FUNCTION "AHUTemperatureDemand" : Void   // FC60007, LAD
{ S7_Optimized_Access := 'TRUE' }
VERSION : 0.1
// stored: AutoNumber false, IsIECCheckEnabled false, SetENOAutomatically false, UDAEnableTagReadback false
   VAR_INPUT
      iUnitID : Int;
      cCoolingRegulatorState : Byte;
      cHeatingRegulatorState : Byte;
      rSATActual : Real;
      rSATSP : Real;
      rRATActual : Real;
      rRATSPHeating : Real;
      rRATSPCooling : Real;
   END_VAR
   VAR_OUTPUT
      rHeatingDemand : Real;
      rCoolingDemand : Real;
      rFreshAirTempDemand : Real;
   END_VAR
   VAR_TEMP
      iActualUnitMode_old : Int;
      xResetActualSetpoints : Bool;
   END_VAR
   VAR CONSTANT
      cZero : Byte;
   END_VAR
   VAR_TEMP   // added for the SCL form of the ladder/FBD networks
      _w1 : Bool;
   END_VAR
BEGIN

REGION Network 1: Cooling
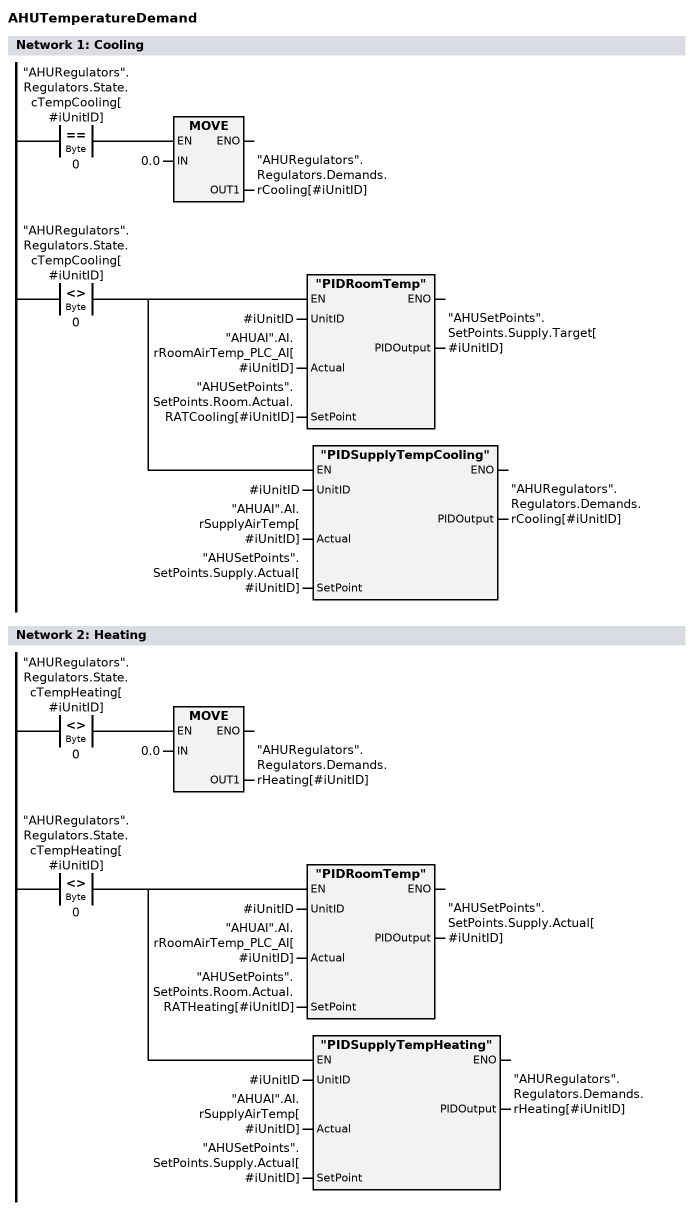
   RUNG wire#powerrail
      { S7_Templates := "SrcType := Byte" } EQ_Contact(in1 := "AHURegulators".Regulators.State.cTempCooling[#iUnitID], in2 := 0)
      Move(in := 0.0, out1 => "AHURegulators".Regulators.Demands.rCooling[#iUnitID])
   END_RUNG
   RUNG wire#powerrail
      { S7_Templates := "SrcType := Byte" } NE_Contact(in1 := "AHURegulators".Regulators.State.cTempCooling[#iUnitID], in2 := 0)
      wire#w1
      "PIDRoomTemp"(UnitID := #iUnitID, Actual := "AHUAI".AI.rRoomAirTemp_PLC_AI[#iUnitID], SetPoint := "AHUSetPoints".SetPoints.Room.Actual.RATCooling[#iUnitID], PIDOutput => "AHUSetPoints".SetPoints.Supply.Target[#iUnitID])
   END_RUNG
   RUNG wire#w1
      "PIDSupplyTempCooling"(UnitID := #iUnitID, Actual := "AHUAI".AI.rSupplyAirTemp[#iUnitID], SetPoint := "AHUSetPoints".SetPoints.Supply.Actual[#iUnitID], PIDOutput => "AHURegulators".Regulators.Demands.rCooling[#iUnitID])
   END_RUNG
   // the same network as SCL:
   IF "AHURegulators".Regulators.State.cTempCooling[#iUnitID] = 0 THEN
       "AHURegulators".Regulators.Demands.rCooling[#iUnitID] := 0.0;
   END_IF;
   #_w1 := "AHURegulators".Regulators.State.cTempCooling[#iUnitID] <> 0;
   IF #_w1 THEN
       "PIDRoomTemp"(UnitID := #iUnitID,
                     Actual := "AHUAI".AI.rRoomAirTemp_PLC_AI[#iUnitID],
                     SetPoint := "AHUSetPoints".SetPoints.Room.Actual.RATCooling[#iUnitID],
                     PIDOutput => "AHUSetPoints".SetPoints.Supply.Target[#iUnitID]);
       "PIDSupplyTempCooling"(UnitID := #iUnitID,
                              Actual := "AHUAI".AI.rSupplyAirTemp[#iUnitID],
                              SetPoint := "AHUSetPoints".SetPoints.Supply.Actual[#iUnitID],
                              PIDOutput => "AHURegulators".Regulators.Demands.rCooling[#iUnitID]);
   END_IF;
END_REGION

REGION Network 2: Heating
   RUNG wire#powerrail
      { S7_Templates := "SrcType := Byte" } NE_Contact(in1 := "AHURegulators".Regulators.State.cTempHeating[#iUnitID], in2 := 0)
      Move(in := 0.0, out1 => "AHURegulators".Regulators.Demands.rHeating[#iUnitID])
   END_RUNG
   RUNG wire#powerrail
      { S7_Templates := "SrcType := Byte" } NE_Contact(in1 := "AHURegulators".Regulators.State.cTempHeating[#iUnitID], in2 := 0)
      wire#w1
      "PIDRoomTemp"(UnitID := #iUnitID, Actual := "AHUAI".AI.rRoomAirTemp_PLC_AI[#iUnitID], SetPoint := "AHUSetPoints".SetPoints.Room.Actual.RATHeating[#iUnitID], PIDOutput => "AHUSetPoints".SetPoints.Supply.Actual[#iUnitID])
   END_RUNG
   RUNG wire#w1
      "PIDSupplyTempHeating"(UnitID := #iUnitID, Actual := "AHUAI".AI.rSupplyAirTemp[#iUnitID], SetPoint := "AHUSetPoints".SetPoints.Supply.Actual[#iUnitID], PIDOutput => "AHURegulators".Regulators.Demands.rHeating[#iUnitID])
   END_RUNG
   // the same network as SCL:
   IF "AHURegulators".Regulators.State.cTempHeating[#iUnitID] <> 0 THEN
       "AHURegulators".Regulators.Demands.rHeating[#iUnitID] := 0.0;
   END_IF;
   #_w1 := "AHURegulators".Regulators.State.cTempHeating[#iUnitID] <> 0;
   IF #_w1 THEN
       "PIDRoomTemp"(UnitID := #iUnitID,
                     Actual := "AHUAI".AI.rRoomAirTemp_PLC_AI[#iUnitID],
                     SetPoint := "AHUSetPoints".SetPoints.Room.Actual.RATHeating[#iUnitID],
                     PIDOutput => "AHUSetPoints".SetPoints.Supply.Actual[#iUnitID]);
       "PIDSupplyTempHeating"(UnitID := #iUnitID,
                              Actual := "AHUAI".AI.rSupplyAirTemp[#iUnitID],
                              SetPoint := "AHUSetPoints".SetPoints.Supply.Actual[#iUnitID],
                              PIDOutput => "AHURegulators".Regulators.Demands.rHeating[#iUnitID]);
   END_IF;
END_REGION
END_FUNCTION

FUNCTION "PIDRoomTemp" : Void   // FC8, FBD
{ S7_Optimized_Access := 'TRUE' }
VERSION : 0.1
// stored: AutoNumber false, IsIECCheckEnabled false, SetENOAutomatically false, UDAEnableTagReadback false
   VAR_INPUT
      UnitID : Int;
      Actual : Real;
      SetPoint : Real;
   END_VAR
   VAR_OUTPUT
      PIDOutput : Real;
   END_VAR
BEGIN
END_FUNCTION

FUNCTION "PIDSupplyTempCooling" : Void   // FC12, FBD
{ S7_Optimized_Access := 'TRUE' }
VERSION : 0.1
// stored: AutoNumber false, IsIECCheckEnabled false, SetENOAutomatically false, UDAEnableTagReadback false
   VAR_INPUT
      UnitID : Int;
      Actual : Real;
      SetPoint : Real;
   END_VAR
   VAR_OUTPUT
      PIDOutput : Real;
   END_VAR
BEGIN
END_FUNCTION

FUNCTION "PIDSupplyTempHeating" : Void   // FC10, FBD
{ S7_Optimized_Access := 'TRUE' }
VERSION : 0.1
// stored: AutoNumber false, IsIECCheckEnabled false, SetENOAutomatically false, UDAEnableTagReadback false
   VAR_INPUT
      UnitID : Int;
      Actual : Real;
      SetPoint : Real;
   END_VAR
   VAR_OUTPUT
      PIDOutput : Real;
   END_VAR
BEGIN
END_FUNCTION

FUNCTION "AHUIAQDemand" : Void   // FC60009, LAD
{ S7_Optimized_Access := 'TRUE' }
VERSION : 0.1
// stored: AutoNumber false, IsIECCheckEnabled false, SetENOAutomatically false, UDAEnableTagReadback false
   VAR_INPUT
      iUnitID : Int;
      cRegState : Byte;
      rActual : Real;
      rSetPoint : Real;
   END_VAR
   VAR_OUTPUT
      rDemand : Real;
   END_VAR
BEGIN
END_FUNCTION

FUNCTION "AHUdPDemand" : Void   // FC60010, LAD
{ S7_Optimized_Access := 'TRUE' }
VERSION : 0.1
// stored: AutoNumber false, IsIECCheckEnabled false, SetENOAutomatically false, UDAEnableTagReadback false
   VAR_INPUT
      iUnitID : Int;
      cRegState : Byte;
      rActual : Real;
      rSetPoint : Real;
   END_VAR
   VAR_OUTPUT
      rDemand : Real;
   END_VAR
BEGIN
END_FUNCTION

FUNCTION "AHUFrostProtectionDemand" : Void   // FC60018, LAD
{ S7_Optimized_Access := 'TRUE' }
VERSION : 0.1
// stored: AutoNumber false, IsIECCheckEnabled false, SetENOAutomatically false, UDAEnableTagReadback false
   VAR_INPUT
      UnitID : Int;
      SupplyAirTemp : Real;
      FrostSensorAirTemp : Real;
      FrostSensorWaterTemp : Real;
      FrostTstat : Bool;
      OutdoorAirTemperature : Real;
   END_VAR
   VAR_OUTPUT
      FrostProtectionDemand : Real;
   END_VAR
BEGIN
END_FUNCTION

FUNCTION "AHU_EqpCtrl" : Void   // FC60300, FBD
{ S7_Optimized_Access := 'TRUE' }
VERSION : 0.1
// stored: AutoNumber false, IsIECCheckEnabled false, SetENOAutomatically false, UDAEnableTagReadback false
   VAR_INPUT
      iUnitID : Int;   // 1=AHUFood, 2=AHUNonFood
   END_VAR
   VAR_TEMP
      FA_temp : Real;
   END_VAR
BEGIN

REGION Network 1: Forming Eqp State with respect of Season and Actual State
   // 0 = Winter
   // 1= Summer
   // 2=Midseason
   // 3=Auto
   // 
   // "HVAC".Season.Actual
   // 0 = Winter
   // 1=Summer
   // 2=Midseason
   // 3=Auto
   // 
   // Type                                             Control State
   // 0 = no ctrl                                             0 = Stopped/Closed/NA
   // 1 = Proxi/Adaptation                           1 = 100%/FullyOpened/ 
   // 2=                                                           2 = RegulationEnable
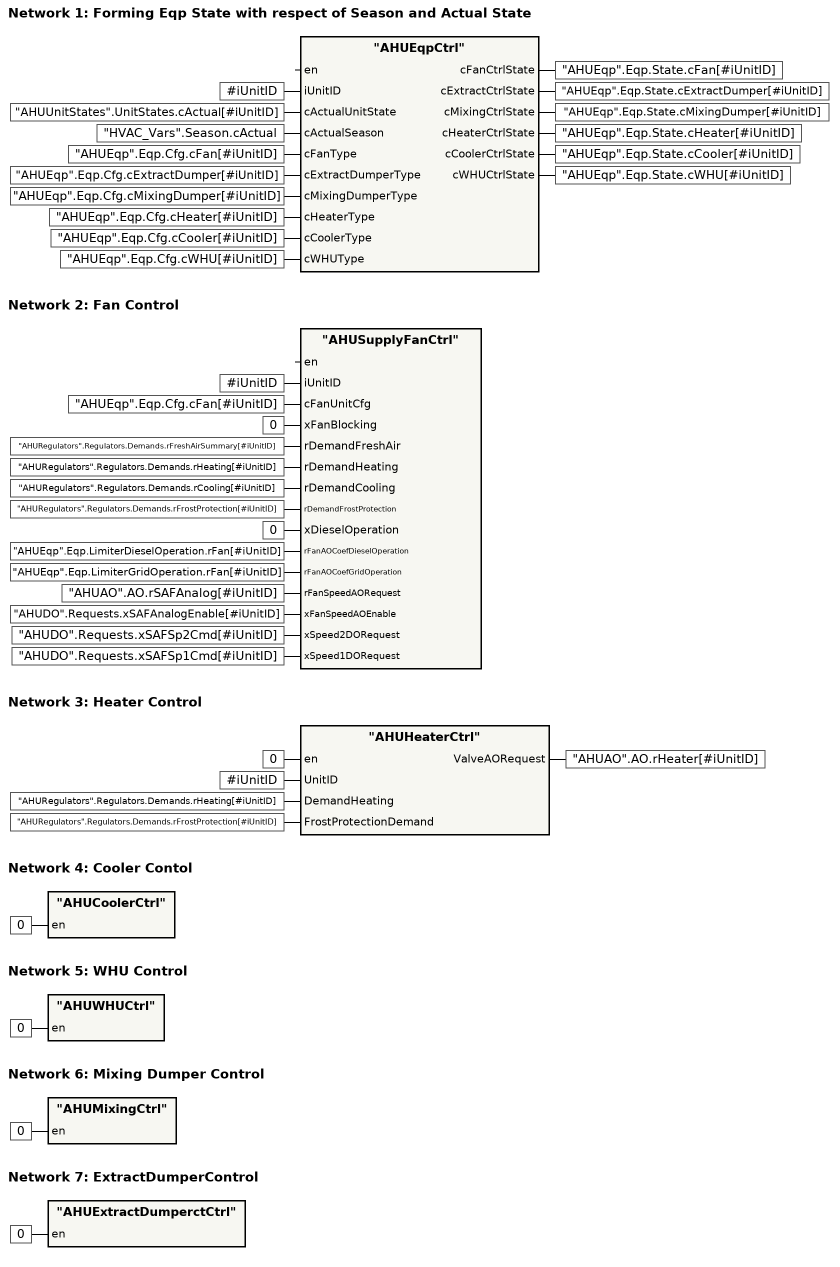
   "AHUEqpCtrl"(iUnitID := #iUnitID,
                cActualUnitState := "AHUUnitStates".UnitStates.cActual[#iUnitID],
                cActualSeason := "HVAC_Vars".Season.cActual,
                cFanType := "AHUEqp".Eqp.Cfg.cFan[#iUnitID],
                cExtractDumperType := "AHUEqp".Eqp.Cfg.cExtractDumper[#iUnitID],
                cMixingDumperType := "AHUEqp".Eqp.Cfg.cMixingDumper[#iUnitID],
                cHeaterType := "AHUEqp".Eqp.Cfg.cHeater[#iUnitID],
                cCoolerType := "AHUEqp".Eqp.Cfg.cCooler[#iUnitID],
                cWHUType := "AHUEqp".Eqp.Cfg.cWHU[#iUnitID],
                cFanCtrlState => "AHUEqp".Eqp.State.cFan[#iUnitID],
                cExtractCtrlState => "AHUEqp".Eqp.State.cExtractDumper[#iUnitID],
                cMixingCtrlState => "AHUEqp".Eqp.State.cMixingDumper[#iUnitID],
                cHeaterCtrlState => "AHUEqp".Eqp.State.cHeater[#iUnitID],
                cCoolerCtrlState => "AHUEqp".Eqp.State.cCooler[#iUnitID],
                cWHUCtrlState => "AHUEqp".Eqp.State.cWHU[#iUnitID]);
END_REGION

REGION Network 2: Fan Control
   "AHUSupplyFanCtrl"(iUnitID := #iUnitID,
                      cFanUnitCfg := "AHUEqp".Eqp.Cfg.cFan[#iUnitID],
                      xFanBlocking := 0,
                      rDemandFreshAir := "AHURegulators".Regulators.Demands.rFreshAirSummary[#iUnitID],
                      rDemandHeating := "AHURegulators".Regulators.Demands.rHeating[#iUnitID],
                      rDemandCooling := "AHURegulators".Regulators.Demands.rCooling[#iUnitID],
                      rDemandFrostProtection := "AHURegulators".Regulators.Demands.rFrostProtection[#iUnitID],
                      xDieselOperation := 0,
                      rFanAOCoefDieselOperation := "AHUEqp".Eqp.LimiterDieselOperation.rFan[#iUnitID],
                      rFanAOCoefGridOperation := "AHUEqp".Eqp.LimiterGridOperation.rFan[#iUnitID],
                      rFanSpeedAORequest := "AHUAO".AO.rSAFAnalog[#iUnitID],
                      xFanSpeedAOEnable := "AHUDO".Requests.xSAFAnalogEnable[#iUnitID],
                      xSpeed2DORequest := "AHUDO".Requests.xSAFSp2Cmd[#iUnitID],
                      xSpeed1DORequest := "AHUDO".Requests.xSAFSp1Cmd[#iUnitID]);
END_REGION

REGION Network 3: Heater Control
   IF 0 THEN
       "AHUHeaterCtrl"(UnitID := #iUnitID,
                       DemandHeating := "AHURegulators".Regulators.Demands.rHeating[#iUnitID],
                       FrostProtectionDemand := "AHURegulators".Regulators.Demands.rFrostProtection[#iUnitID],
                       ValveAORequest => "AHUAO".AO.rHeater[#iUnitID]);
   END_IF;
END_REGION

REGION Network 4: Cooler Contol
   IF 0 THEN "AHUCoolerCtrl"(); END_IF;
END_REGION

REGION Network 5: WHU Control
   IF 0 THEN "AHUWHUCtrl"(); END_IF;
END_REGION

REGION Network 6: Mixing Dumper Control
   IF 0 THEN "AHUMixingCtrl"(); END_IF;
END_REGION

REGION Network 7: ExtractDumperControl
   IF 0 THEN "AHUExtractDumperctCtrl"(); END_IF;
END_REGION
END_FUNCTION

FUNCTION "AHUEqpCtrl" : Void   // FC60301, LAD
{ S7_Optimized_Access := 'TRUE' }
VERSION : 0.1
// Type                                             Control State
// 0 = no ctrl                                             0 = Stopped/Closed/NA
// 1 = Proxi/Adaptation                           1 = 100%/FullyOpened/ 
// 2=                                                           2 = RegulationEnable
// stored: AutoNumber false, IsIECCheckEnabled false, SetENOAutomatically false, UDAEnableTagReadback false
   VAR_INPUT
      iUnitID : Int;
      cActualUnitState : Byte;
      cActualSeason : Byte;
      cFanType : Byte;
      cExtractDumperType : Byte;
      cMixingDumperType : Byte;
      cHeaterType : Byte;
      cCoolerType : Byte;
      cWHUType : Byte;
   END_VAR
   VAR_OUTPUT
      cFanCtrlState : Byte;
      cExtractCtrlState : Byte;
      cMixingCtrlState : Byte;
      cHeaterCtrlState : Byte;
      cCoolerCtrlState : Byte;
      cWHUCtrlState : Byte;
   END_VAR
BEGIN

REGION Network 1 (SCL): Fan
   CASE #cFanType OF
       0:  //disable
           #cFanCtrlState := 0;
       ELSE  // Active
           #cFanCtrlState := 2;
   END_CASE;
END_REGION

REGION Network 2 (SCL): Extract Dumper
   CASE #cExtractDumperType OF
       0:  //disable
           #cExtractCtrlState := 0;
       ELSE  // Active
           CASE #cActualSeason OF
               0:  // Winter
                   #cExtractCtrlState := 0;//Blocked
               1:  // Summer
                   #cExtractCtrlState := 0;//Auto
               ELSE  //Midseason
                   #cExtractCtrlState := 2;//Auto
           END_CASE;
   END_CASE;
END_REGION

REGION Network 3 (SCL): Mixing Dumper
   CASE #cMixingDumperType OF
       0:  //disable
           #cMixingCtrlState := 0;
       ELSE  // Active
           IF #cActualUnitState = 4 THEN // 100% recycling mode
               #cMixingCtrlState := 1;
           ELSE
               #cMixingCtrlState := 2;
           END_IF;
   END_CASE;
END_REGION

REGION Network 4 (SCL): Heater
   CASE #cHeaterType OF
       0:  //disable
           #cHeaterCtrlState := 0;
       ELSE  // Active
           IF #cActualUnitState =2  THEN //Preheating
               #cHeaterCtrlState := 1;
           ELSE

               CASE #cActualSeason OF
                   0:  // Winter
                       #cHeaterCtrlState := 2;//Auto
                   1:  // Summer
                       #cHeaterCtrlState := 0;//Blocked
                   ELSE  //Midseason
                       #cHeaterCtrlState := 2;//Auto
               END_CASE;
           END_IF;
   END_CASE;
END_REGION

REGION Network 5 (SCL): Cooler
   CASE #cCoolerType OF
       0:  //disable
           #cCoolerCtrlState := 0;
       ELSE  // Active
           CASE #cActualSeason OF
               0:  //Winter
                   #cCoolerCtrlState := 0;//Blocked
               1:  // Summer
                   #cCoolerCtrlState := 2;//Auto
               ELSE  //Midseason
                   #cCoolerCtrlState := 2;//Auto
           END_CASE;
   END_CASE;
END_REGION

REGION Network 6 (SCL): WHU
   CASE #cWHUType OF
       0:  //disable
           #cWHUCtrlState := 0;
       ELSE  // Active
           CASE #cActualSeason OF
               0:  // Winter
                   #cWHUCtrlState := 2;//Auto
               1:  // Summer
                   #cWHUCtrlState := 0;//Blocked
               ELSE  //Midseason
                   #cWHUCtrlState := 2;//Auto
           END_CASE;
   END_CASE;
END_REGION
END_FUNCTION

FUNCTION "AHUSupplyFanCtrl" : Void   // FC60302, LAD
{ S7_Optimized_Access := 'TRUE' }
VERSION : 0.1
// Cfg
// 0 - No Fan (No AHU)
// 1 - Adaptation/Proxi
// 2 - 1Speed
// 3 - 2Speed
// 4 - 0-100%
// stored: AutoNumber false, IsIECCheckEnabled false, SetENOAutomatically false, UDAEnableTagReadback false
   VAR_INPUT
      iUnitID : Int;
      cFanUnitCfg : Byte;
      xFanBlocking : Bool;
      rDemandFreshAir : Real;
      rDemandHeating : Real;
      rDemandCooling : Real;
      rDemandFrostProtection : Real;
      xDieselOperation : Bool;
      rFanAOCoefDieselOperation : Real;
      rFanAOCoefGridOperation : Real;
   END_VAR
   VAR_IN_OUT
      rFanSpeedAORequest : Real;
      xFanSpeedAOEnable : Bool;
      xSpeed2DORequest : Bool;
      xSpeed1DORequest : Bool;
   END_VAR
   VAR_TEMP
      rSumDemand : Real;
      rSumDemandInt1 : Real;
      rSumDemandInt2 : Real;
      rRawFanAO : Real;
      xRawFanSt1Request : Bool;
      xRawFanSt2Request : Bool;
      xRawFanAOEnable : Bool;
   END_VAR
BEGIN

REGION Network 1 (SCL)
   CASE #cFanUnitCfg OF
       0:  // No Unit
           ;
       1:  // Proxy
           ;
       2:   // Single speed
           ; 
       3:   // Two speed fan motor
           ;
       4:  // 0-100% Modulative
           #xSpeed1DORequest := 0;
           #xSpeed2DORequest := 0;

           IF #xFanBlocking THEN
               #rRawFanAO := 0;
               #xFanSpeedAOEnable := 0;
           ELSE
               #rSumDemandInt1 := MAX(IN1 := #rDemandFreshAir, IN2 := #rDemandHeating);
               #rSumDemandInt2 := MAX(IN1 := #rDemandFrostProtection, IN2 := #rDemandCooling);
               #rSumDemand := MAX(IN1 := #rSumDemandInt1, IN2 := #rSumDemandInt2);

               IF #rSumDemand > 5 THEN
                   #rFanSpeedAORequest := 1;
                   #rRawFanAO := #rSumDemand;
               ELSIF #rSumDemand < 1 THEN
                   #rFanSpeedAORequest := 0;
                   #xFanSpeedAOEnable := 0;
               END_IF;
           END_IF;
           ;
       ELSE  // Statement section ELSE
           ;
   END_CASE;
END_REGION

REGION Network 2 (SCL)
   IF #xDieselOperation THEN
       #xSpeed2DORequest := 0;
       #xSpeed1DORequest := #xRawFanSt1Request OR #xRawFanSt2Request;
       #rFanSpeedAORequest := #rRawFanAO * #rFanAOCoefDieselOperation;
       #xFanSpeedAOEnable := #xRawFanAOEnable;
   END_IF;
END_REGION
END_FUNCTION

FUNCTION "AHUHeaterCtrl" : Void   // FC60303, LAD
{ S7_Optimized_Access := 'TRUE' }
VERSION : 0.1
// stored: AutoNumber false, IsIECCheckEnabled false, SetENOAutomatically false, UDAEnableTagReadback false
   VAR_INPUT
      UnitID : Int;
      DemandHeating : Real;
      FrostProtectionDemand : Real;
   END_VAR
   VAR_OUTPUT
      ValveAORequest : Real;
   END_VAR
BEGIN
END_FUNCTION

FUNCTION "AHUCoolerCtrl" : Void   // FC60304, LAD
{ S7_Optimized_Access := 'TRUE' }
VERSION : 0.1
// stored: AutoNumber false, IsIECCheckEnabled false, SetENOAutomatically false, UDAEnableTagReadback false
BEGIN
END_FUNCTION

FUNCTION "AHUWHUCtrl" : Void   // FC60305, LAD
{ S7_Optimized_Access := 'TRUE' }
VERSION : 0.1
// stored: AutoNumber false, IsIECCheckEnabled false, SetENOAutomatically false, UDAEnableTagReadback false
BEGIN
END_FUNCTION

FUNCTION "AHUMixingCtrl" : Void   // FC60306, LAD
{ S7_Optimized_Access := 'TRUE' }
VERSION : 0.1
// stored: AutoNumber false, IsIECCheckEnabled false, SetENOAutomatically false, UDAEnableTagReadback false
BEGIN
END_FUNCTION

FUNCTION "AHUExtractDumperctCtrl" : Void   // FC60307, LAD
{ S7_Optimized_Access := 'TRUE' }
VERSION : 0.1
// stored: AutoNumber false, IsIECCheckEnabled false, SetENOAutomatically false, UDAEnableTagReadback false
BEGIN
END_FUNCTION

FUNCTION "DL_General" : Void   // FC51001, LAD
{ S7_Optimized_Access := 'TRUE' }
VERSION : 0.1
// stored: AutoNumber false, IsIECCheckEnabled false, SetENOAutomatically false, UDAEnableTagReadback false
   VAR_TEMP
      LvlRequest : Array[1..2] of Bool;
      xStopTriger : Bool;
      xCounter1Triger : Bool;
      xCounter2Triger : Bool;
      xPump1ExeriseRun : Bool;
      xPump2ExeriseRun : Bool;
      xPump1ExeriseRunTriger : Bool;
      xPump2ExeriseRunTriger : Bool;
      tTimeExericePump1 : Time;
      tTimeExericePump2 : Time;
   END_VAR
   VAR_TEMP   // added for the SCL form of the ladder/FBD networks
      _w1 : Bool;
      _w2 : Bool;
      _w3 : Bool;
      _w4 : Bool;
      _w5 : Bool;
      _w6 : Bool;
   END_VAR
BEGIN

REGION Network 1 (SCL): PanelModeSelector
   IF "DLsDI".Requests.xDieselLinePumpPanelSelectorAuto THEN
       "DL_Vars".Vars.cDLPanelModeSelector := 3;
   ELSIF "DLsDI".Requests.xDieselLinePumpPanelSelectorP1Man THEN
       "DL_Vars".Vars.cDLPanelModeSelector := 1;
   ELSIF "DLsDI".Requests.xDieselLinePumpPanelSelectorP2Man THEN
       "DL_Vars".Vars.cDLPanelModeSelector := 2;
   ELSIF "DLsDI".Requests.xDieselLinePumpPanelSelectorOff THEN
       "DL_Vars".Vars.cDLPanelModeSelector := 0;
   END_IF;
END_REGION

REGION Network 2
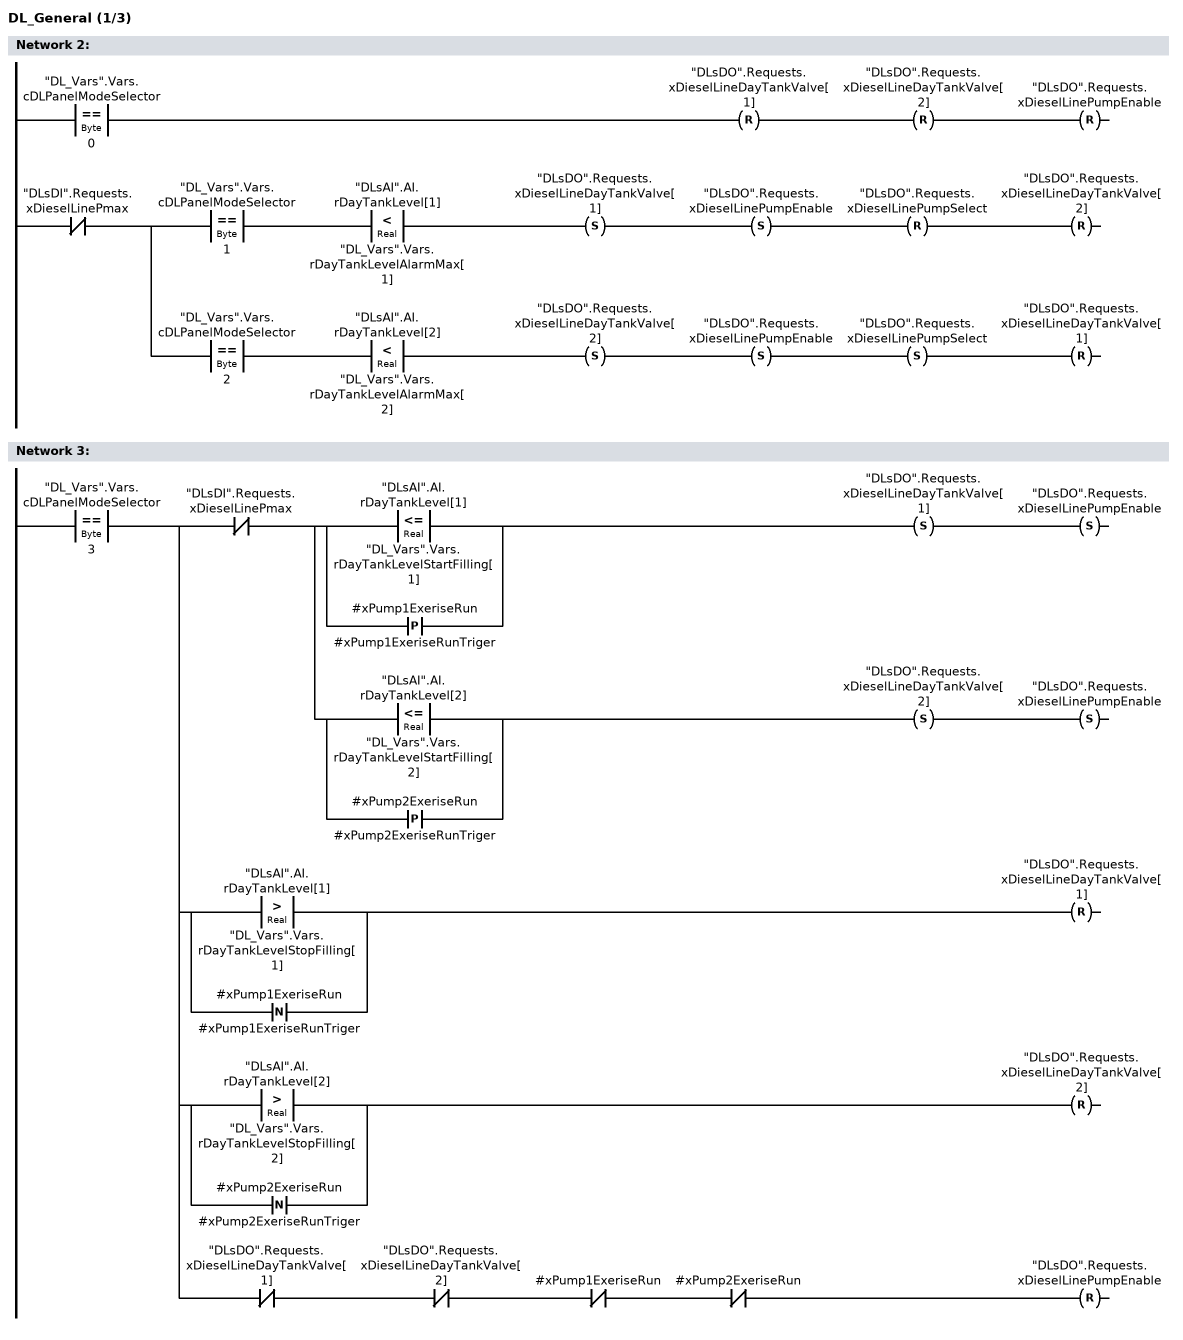
   RUNG wire#powerrail
      { S7_Templates := "SrcType := Byte" } EQ_Contact(in1 := "DL_Vars".Vars.cDLPanelModeSelector, in2 := 0)
      R_Coil( "DLsDO".Requests.xDieselLineDayTankValve[1] )
      R_Coil( "DLsDO".Requests.xDieselLineDayTankValve[2] )
      R_Coil( "DLsDO".Requests.xDieselLinePumpEnable )
   END_RUNG
   RUNG wire#powerrail
      I_Contact( "DLsDI".Requests.xDieselLinePmax )
      wire#w1
      { S7_Templates := "SrcType := Byte" } EQ_Contact(in1 := "DL_Vars".Vars.cDLPanelModeSelector, in2 := 1)
      { S7_Templates := "SrcType := Real" } LT_Contact(in1 := "DLsAI".AI.rDayTankLevel[1], in2 := "DL_Vars".Vars.rDayTankLevelAlarmMax[1])
      S_Coil( "DLsDO".Requests.xDieselLineDayTankValve[1] )
      S_Coil( "DLsDO".Requests.xDieselLinePumpEnable )
      R_Coil( "DLsDO".Requests.xDieselLinePumpSelect )
      R_Coil( "DLsDO".Requests.xDieselLineDayTankValve[2] )
   END_RUNG
   RUNG wire#w1
      { S7_Templates := "SrcType := Byte" } EQ_Contact(in1 := "DL_Vars".Vars.cDLPanelModeSelector, in2 := 2)
      { S7_Templates := "SrcType := Real" } LT_Contact(in1 := "DLsAI".AI.rDayTankLevel[2], in2 := "DL_Vars".Vars.rDayTankLevelAlarmMax[2])
      S_Coil( "DLsDO".Requests.xDieselLineDayTankValve[2] )
      S_Coil( "DLsDO".Requests.xDieselLinePumpEnable )
      S_Coil( "DLsDO".Requests.xDieselLinePumpSelect )
      R_Coil( "DLsDO".Requests.xDieselLineDayTankValve[1] )
   END_RUNG
   // the same network as SCL:
   IF "DL_Vars".Vars.cDLPanelModeSelector = 0 THEN
       "DLsDO".Requests.xDieselLineDayTankValve[1] := FALSE;
       "DLsDO".Requests.xDieselLineDayTankValve[2] := FALSE;
       "DLsDO".Requests.xDieselLinePumpEnable := FALSE;
   END_IF;
   #_w1 := NOT "DLsDI".Requests.xDieselLinePmax;
   IF #_w1 AND ("DL_Vars".Vars.cDLPanelModeSelector = 1) AND ("DLsAI".AI.rDayTankLevel[1] < "DL_Vars".Vars.rDayTankLevelAlarmMax[1]) THEN
       "DLsDO".Requests.xDieselLineDayTankValve[1] := TRUE;
       "DLsDO".Requests.xDieselLinePumpEnable := TRUE;
       "DLsDO".Requests.xDieselLinePumpSelect := FALSE;
       "DLsDO".Requests.xDieselLineDayTankValve[2] := FALSE;
   END_IF;
   IF #_w1 AND ("DL_Vars".Vars.cDLPanelModeSelector = 2) AND ("DLsAI".AI.rDayTankLevel[2] < "DL_Vars".Vars.rDayTankLevelAlarmMax[2]) THEN
       "DLsDO".Requests.xDieselLineDayTankValve[2] := TRUE;
       "DLsDO".Requests.xDieselLinePumpEnable := TRUE;
       "DLsDO".Requests.xDieselLinePumpSelect := TRUE;
       "DLsDO".Requests.xDieselLineDayTankValve[1] := FALSE;
   END_IF;
END_REGION

REGION Network 3
   RUNG wire#powerrail
      { S7_Templates := "SrcType := Byte" } EQ_Contact(in1 := "DL_Vars".Vars.cDLPanelModeSelector, in2 := 3)
      wire#w1
      I_Contact( "DLsDI".Requests.xDieselLinePmax )
      wire#w2
      { S7_Templates := "SrcType := Real" } LE_Contact(in1 := "DLsAI".AI.rDayTankLevel[1], in2 := "DL_Vars".Vars.rDayTankLevelStartFilling[1])
      wire#w3
      S_Coil( "DLsDO".Requests.xDieselLineDayTankValve[1] )
      S_Coil( "DLsDO".Requests.xDieselLinePumpEnable )
   END_RUNG
   RUNG wire#w2
      P_Contact(operand := #xPump1ExeriseRun, bit := #xPump1ExeriseRunTriger)
   END_RUNG wire#w3
   RUNG wire#w2
      { S7_Templates := "SrcType := Real" } LE_Contact(in1 := "DLsAI".AI.rDayTankLevel[2], in2 := "DL_Vars".Vars.rDayTankLevelStartFilling[2])
      wire#w4
      S_Coil( "DLsDO".Requests.xDieselLineDayTankValve[2] )
      S_Coil( "DLsDO".Requests.xDieselLinePumpEnable )
   END_RUNG
   RUNG wire#w2
      P_Contact(operand := #xPump2ExeriseRun, bit := #xPump2ExeriseRunTriger)
   END_RUNG wire#w4
   RUNG wire#w1
      { S7_Templates := "SrcType := Real" } GT_Contact(in1 := "DLsAI".AI.rDayTankLevel[1], in2 := "DL_Vars".Vars.rDayTankLevelStopFilling[1])
      wire#w5
      R_Coil( "DLsDO".Requests.xDieselLineDayTankValve[1] )
   END_RUNG
   RUNG wire#w1
      N_Contact(operand := #xPump1ExeriseRun, bit := #xPump1ExeriseRunTriger)
   END_RUNG wire#w5
   RUNG wire#w1
      { S7_Templates := "SrcType := Real" } GT_Contact(in1 := "DLsAI".AI.rDayTankLevel[2], in2 := "DL_Vars".Vars.rDayTankLevelStopFilling[2])
      wire#w6
      R_Coil( "DLsDO".Requests.xDieselLineDayTankValve[2] )
   END_RUNG
   RUNG wire#w1
      N_Contact(operand := #xPump2ExeriseRun, bit := #xPump2ExeriseRunTriger)
   END_RUNG wire#w6
   RUNG wire#w1
      I_Contact( "DLsDO".Requests.xDieselLineDayTankValve[1] )
      I_Contact( "DLsDO".Requests.xDieselLineDayTankValve[2] )
      I_Contact( #xPump1ExeriseRun )
      I_Contact( #xPump2ExeriseRun )
      R_Coil( "DLsDO".Requests.xDieselLinePumpEnable )
   END_RUNG
   // the same network as SCL:
   #_w1 := "DL_Vars".Vars.cDLPanelModeSelector = 3;
   #_w2 := #_w1 AND NOT "DLsDI".Requests.xDieselLinePmax;
   #_w3 := #_w2 AND #xPump1ExeriseRun AND NOT #xPump1ExeriseRunTriger;   // rising edge of #xPump1ExeriseRun
   #xPump1ExeriseRunTriger := #xPump1ExeriseRun;
   IF (#_w2 AND ("DLsAI".AI.rDayTankLevel[1] <= "DL_Vars".Vars.rDayTankLevelStartFilling[1])) OR #_w3 THEN
       "DLsDO".Requests.xDieselLineDayTankValve[1] := TRUE;
       "DLsDO".Requests.xDieselLinePumpEnable := TRUE;
   END_IF;
   #_w4 := #_w2 AND #xPump2ExeriseRun AND NOT #xPump2ExeriseRunTriger;   // rising edge of #xPump2ExeriseRun
   #xPump2ExeriseRunTriger := #xPump2ExeriseRun;
   IF (#_w2 AND ("DLsAI".AI.rDayTankLevel[2] <= "DL_Vars".Vars.rDayTankLevelStartFilling[2])) OR #_w4 THEN
       "DLsDO".Requests.xDieselLineDayTankValve[2] := TRUE;
       "DLsDO".Requests.xDieselLinePumpEnable := TRUE;
   END_IF;
   #_w5 := #_w1 AND NOT #xPump1ExeriseRun AND #xPump1ExeriseRunTriger;   // falling edge of #xPump1ExeriseRun
   #xPump1ExeriseRunTriger := #xPump1ExeriseRun;
   IF (#_w1 AND ("DLsAI".AI.rDayTankLevel[1] > "DL_Vars".Vars.rDayTankLevelStopFilling[1])) OR #_w5 THEN
       "DLsDO".Requests.xDieselLineDayTankValve[1] := FALSE;
   END_IF;
   #_w6 := #_w1 AND NOT #xPump2ExeriseRun AND #xPump2ExeriseRunTriger;   // falling edge of #xPump2ExeriseRun
   #xPump2ExeriseRunTriger := #xPump2ExeriseRun;
   IF (#_w1 AND ("DLsAI".AI.rDayTankLevel[2] > "DL_Vars".Vars.rDayTankLevelStopFilling[2])) OR #_w6 THEN
       "DLsDO".Requests.xDieselLineDayTankValve[2] := FALSE;
   END_IF;
   IF #_w1 AND NOT "DLsDO".Requests.xDieselLineDayTankValve[1] AND NOT "DLsDO".Requests.xDieselLineDayTankValve[2] AND NOT #xPump1ExeriseRun AND NOT #xPump2ExeriseRun THEN
       "DLsDO".Requests.xDieselLinePumpEnable := FALSE;
   END_IF;
END_REGION

REGION Network 4
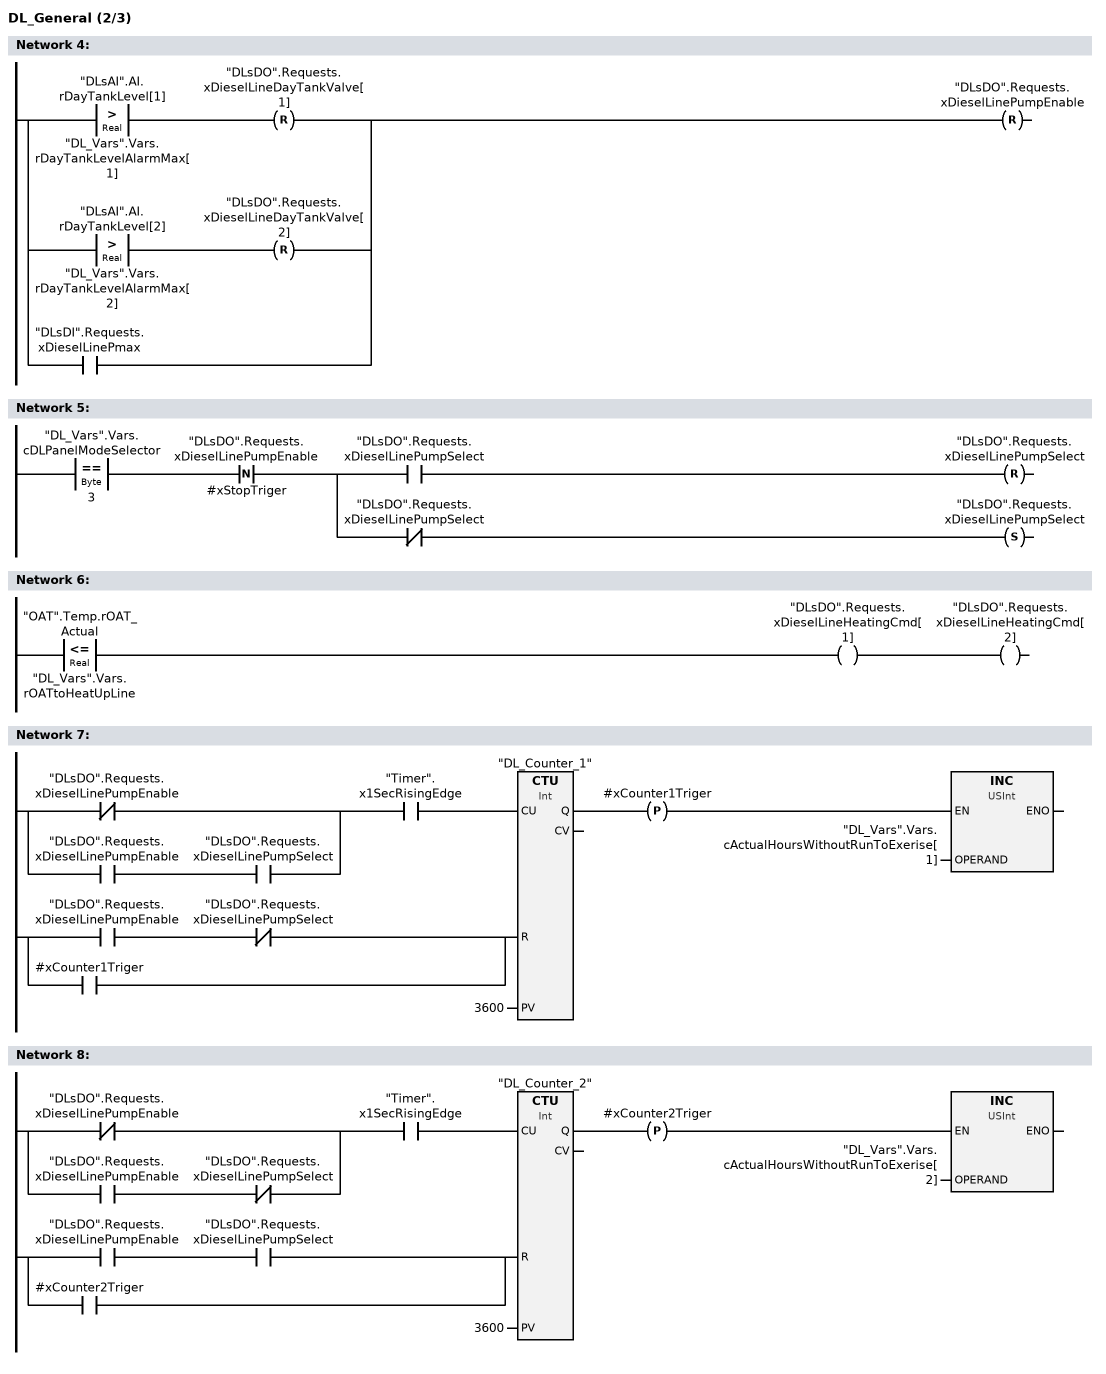
   RUNG wire#powerrail
      { S7_Templates := "SrcType := Real" } GT_Contact(in1 := "DLsAI".AI.rDayTankLevel[1], in2 := "DL_Vars".Vars.rDayTankLevelAlarmMax[1])
      R_Coil( "DLsDO".Requests.xDieselLineDayTankValve[1] )
      wire#w1
      R_Coil( "DLsDO".Requests.xDieselLinePumpEnable )
   END_RUNG
   RUNG wire#powerrail
      { S7_Templates := "SrcType := Real" } GT_Contact(in1 := "DLsAI".AI.rDayTankLevel[2], in2 := "DL_Vars".Vars.rDayTankLevelAlarmMax[2])
      R_Coil( "DLsDO".Requests.xDieselLineDayTankValve[2] )
   END_RUNG wire#w1
   RUNG wire#powerrail
      Contact( "DLsDI".Requests.xDieselLinePmax )
   END_RUNG wire#w1
   // the same network as SCL:
   #_w1 := "DLsAI".AI.rDayTankLevel[1] > "DL_Vars".Vars.rDayTankLevelAlarmMax[1];
   IF #_w1 THEN "DLsDO".Requests.xDieselLineDayTankValve[1] := FALSE; END_IF;
   #_w2 := "DLsAI".AI.rDayTankLevel[2] > "DL_Vars".Vars.rDayTankLevelAlarmMax[2];
   IF #_w2 THEN "DLsDO".Requests.xDieselLineDayTankValve[2] := FALSE; END_IF;
   IF #_w1 OR #_w2 OR "DLsDI".Requests.xDieselLinePmax THEN
       "DLsDO".Requests.xDieselLinePumpEnable := FALSE;
   END_IF;
END_REGION

REGION Network 5
   RUNG wire#powerrail
      { S7_Templates := "SrcType := Byte" } EQ_Contact(in1 := "DL_Vars".Vars.cDLPanelModeSelector, in2 := 3)
      N_Contact(operand := "DLsDO".Requests.xDieselLinePumpEnable, bit := #xStopTriger)
      wire#w1
      Contact( "DLsDO".Requests.xDieselLinePumpSelect )
      R_Coil( "DLsDO".Requests.xDieselLinePumpSelect )
   END_RUNG
   RUNG wire#w1
      I_Contact( "DLsDO".Requests.xDieselLinePumpSelect )
      S_Coil( "DLsDO".Requests.xDieselLinePumpSelect )
   END_RUNG
   // the same network as SCL:
   #_w1 := ("DL_Vars".Vars.cDLPanelModeSelector = 3) AND NOT "DLsDO".Requests.xDieselLinePumpEnable AND #xStopTriger;   // falling edge of "DLsDO".Requests.xDieselLinePumpEnable
   #xStopTriger := "DLsDO".Requests.xDieselLinePumpEnable;
   IF #_w1 AND "DLsDO".Requests.xDieselLinePumpSelect THEN
       "DLsDO".Requests.xDieselLinePumpSelect := FALSE;
   END_IF;
   IF #_w1 AND NOT "DLsDO".Requests.xDieselLinePumpSelect THEN
       "DLsDO".Requests.xDieselLinePumpSelect := TRUE;
   END_IF;
END_REGION

REGION Network 6
   RUNG wire#powerrail
      { S7_Templates := "SrcType := Real" } LE_Contact(in1 := "OAT".Temp.rOAT_Actual, in2 := "DL_Vars".Vars.rOATtoHeatUpLine)
      Coil( "DLsDO".Requests.xDieselLineHeatingCmd[1] )
      Coil( "DLsDO".Requests.xDieselLineHeatingCmd[2] )
   END_RUNG
   // the same network as SCL:
   "DLsDO".Requests.xDieselLineHeatingCmd[1] := "OAT".Temp.rOAT_Actual <= "DL_Vars".Vars.rOATtoHeatUpLine;
   "DLsDO".Requests.xDieselLineHeatingCmd[2] := "OAT".Temp.rOAT_Actual <= "DL_Vars".Vars.rOATtoHeatUpLine;
END_REGION

REGION Network 7
   RUNG wire#powerrail
      I_Contact( "DLsDO".Requests.xDieselLinePumpEnable )
      wire#w1
      Contact( "Timer".x1SecRisingEdge )
      { S7_Templates := "value_type := Int" } "DL_Counter_1".CTU(r := wire#w2, pv := 3600, cv =>)
      P_Trig( #xCounter1Triger )
      { S7_Templates := "DestType := USInt" } Inc( "DL_Vars".Vars.cActualHoursWithoutRunToExerise[1] )
   END_RUNG
   RUNG wire#powerrail
      Contact( "DLsDO".Requests.xDieselLinePumpEnable )
      Contact( "DLsDO".Requests.xDieselLinePumpSelect )
   END_RUNG wire#w1
   RUNG wire#powerrail
      Contact( "DLsDO".Requests.xDieselLinePumpEnable )
      I_Contact( "DLsDO".Requests.xDieselLinePumpSelect )
   END_RUNG wire#w2
   RUNG wire#powerrail
      Contact( #xCounter1Triger )
   END_RUNG wire#w2
   // the same network as SCL:
   "DL_Counter_1".CTU(CU := (NOT "DLsDO".Requests.xDieselLinePumpEnable OR ("DLsDO".Requests.xDieselLinePumpEnable AND "DLsDO".Requests.xDieselLinePumpSelect)) AND "Timer".x1SecRisingEdge,
                      R := ("DLsDO".Requests.xDieselLinePumpEnable AND NOT "DLsDO".Requests.xDieselLinePumpSelect) OR #xCounter1Triger,
                      PV := 3600);
   #_w1 := "DL_Counter_1".Q AND NOT #xCounter1Triger;   // rising edge
   #xCounter1Triger := "DL_Counter_1".Q;
   IF #_w1 THEN
       "DL_Vars".Vars.cActualHoursWithoutRunToExerise[1] := "DL_Vars".Vars.cActualHoursWithoutRunToExerise[1] + 1;
   END_IF;
END_REGION

REGION Network 8
   RUNG wire#powerrail
      I_Contact( "DLsDO".Requests.xDieselLinePumpEnable )
      wire#w1
      Contact( "Timer".x1SecRisingEdge )
      { S7_Templates := "value_type := Int" } "DL_Counter_2".CTU(r := wire#w2, pv := 3600, cv =>)
      P_Trig( #xCounter2Triger )
      { S7_Templates := "DestType := USInt" } Inc( "DL_Vars".Vars.cActualHoursWithoutRunToExerise[2] )
   END_RUNG
   RUNG wire#powerrail
      Contact( "DLsDO".Requests.xDieselLinePumpEnable )
      I_Contact( "DLsDO".Requests.xDieselLinePumpSelect )
   END_RUNG wire#w1
   RUNG wire#powerrail
      Contact( "DLsDO".Requests.xDieselLinePumpEnable )
      Contact( "DLsDO".Requests.xDieselLinePumpSelect )
   END_RUNG wire#w2
   RUNG wire#powerrail
      Contact( #xCounter2Triger )
   END_RUNG wire#w2
   // the same network as SCL:
   "DL_Counter_2".CTU(CU := (NOT "DLsDO".Requests.xDieselLinePumpEnable OR ("DLsDO".Requests.xDieselLinePumpEnable AND NOT "DLsDO".Requests.xDieselLinePumpSelect)) AND "Timer".x1SecRisingEdge,
                      R := ("DLsDO".Requests.xDieselLinePumpEnable AND "DLsDO".Requests.xDieselLinePumpSelect) OR #xCounter2Triger,
                      PV := 3600);
   #_w1 := "DL_Counter_2".Q AND NOT #xCounter2Triger;   // rising edge
   #xCounter2Triger := "DL_Counter_2".Q;
   IF #_w1 THEN
       "DL_Vars".Vars.cActualHoursWithoutRunToExerise[2] := "DL_Vars".Vars.cActualHoursWithoutRunToExerise[2] + 1;
   END_IF;
END_REGION

REGION Network 9
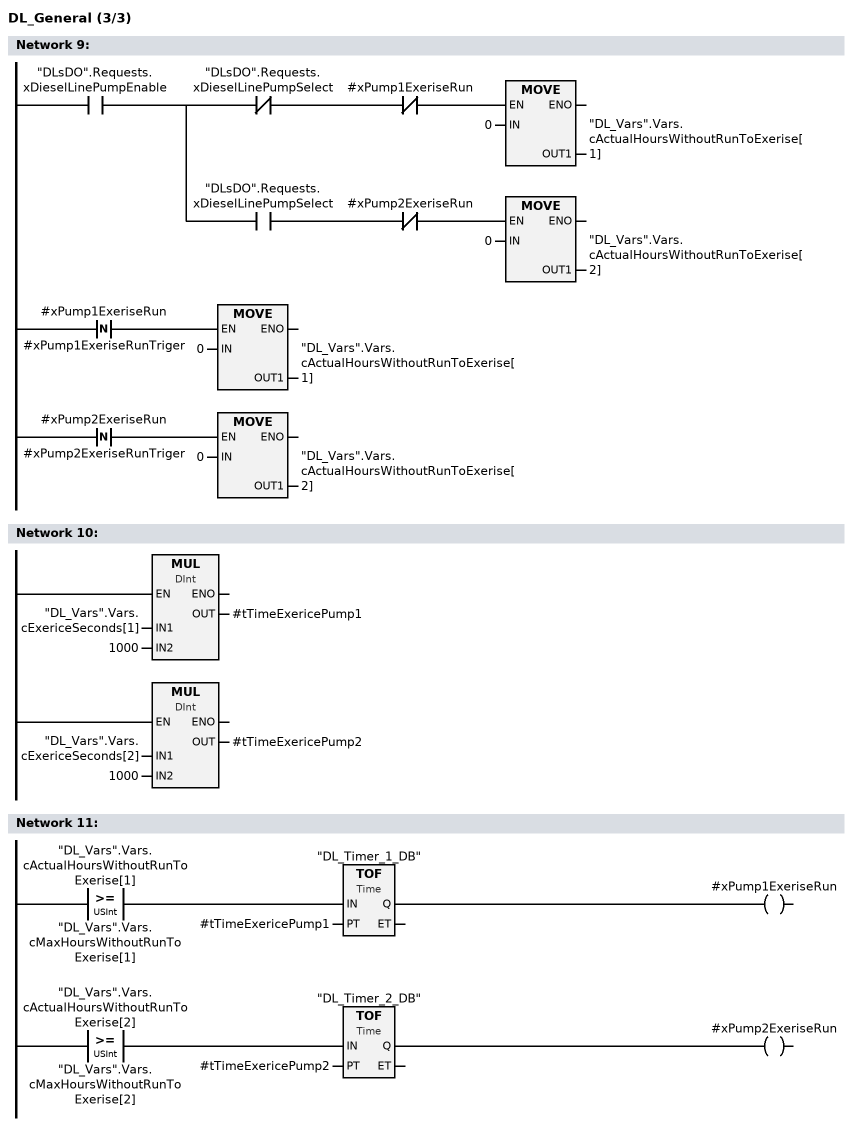
   RUNG wire#powerrail
      Contact( "DLsDO".Requests.xDieselLinePumpEnable )
      wire#w1
      I_Contact( "DLsDO".Requests.xDieselLinePumpSelect )
      I_Contact( #xPump1ExeriseRun )
      Move(in := 0, out1 => "DL_Vars".Vars.cActualHoursWithoutRunToExerise[1])
   END_RUNG
   RUNG wire#w1
      Contact( "DLsDO".Requests.xDieselLinePumpSelect )
      I_Contact( #xPump2ExeriseRun )
      Move(in := 0, out1 => "DL_Vars".Vars.cActualHoursWithoutRunToExerise[2])
   END_RUNG
   RUNG wire#powerrail
      N_Contact(operand := #xPump1ExeriseRun, bit := #xPump1ExeriseRunTriger)
      Move(in := 0, out1 => "DL_Vars".Vars.cActualHoursWithoutRunToExerise[1])
   END_RUNG
   RUNG wire#powerrail
      N_Contact(operand := #xPump2ExeriseRun, bit := #xPump2ExeriseRunTriger)
      Move(in := 0, out1 => "DL_Vars".Vars.cActualHoursWithoutRunToExerise[2])
   END_RUNG
   // the same network as SCL:
   IF "DLsDO".Requests.xDieselLinePumpEnable AND NOT "DLsDO".Requests.xDieselLinePumpSelect AND NOT #xPump1ExeriseRun THEN
       "DL_Vars".Vars.cActualHoursWithoutRunToExerise[1] := 0;
   END_IF;
   IF "DLsDO".Requests.xDieselLinePumpEnable AND "DLsDO".Requests.xDieselLinePumpSelect AND NOT #xPump2ExeriseRun THEN
       "DL_Vars".Vars.cActualHoursWithoutRunToExerise[2] := 0;
   END_IF;
   #_w1 := NOT #xPump1ExeriseRun AND #xPump1ExeriseRunTriger;   // falling edge of #xPump1ExeriseRun
   #xPump1ExeriseRunTriger := #xPump1ExeriseRun;
   IF #_w1 THEN "DL_Vars".Vars.cActualHoursWithoutRunToExerise[1] := 0; END_IF;
   #_w2 := NOT #xPump2ExeriseRun AND #xPump2ExeriseRunTriger;   // falling edge of #xPump2ExeriseRun
   #xPump2ExeriseRunTriger := #xPump2ExeriseRun;
   IF #_w2 THEN "DL_Vars".Vars.cActualHoursWithoutRunToExerise[2] := 0; END_IF;
END_REGION

REGION Network 10
   RUNG wire#powerrail
      { S7_Templates := "SrcType := DInt" } Mul(in1 := "DL_Vars".Vars.cExericeSeconds[1], in2 := 1000, out => #tTimeExericePump1)
   END_RUNG
   RUNG wire#powerrail
      { S7_Templates := "SrcType := DInt" } Mul(in1 := "DL_Vars".Vars.cExericeSeconds[2], in2 := 1000, out => #tTimeExericePump2)
   END_RUNG
   // the same network as SCL:
   #tTimeExericePump1 := "DL_Vars".Vars.cExericeSeconds[1] * 1000;
   #tTimeExericePump2 := "DL_Vars".Vars.cExericeSeconds[2] * 1000;
END_REGION

REGION Network 11
   RUNG wire#powerrail
      { S7_Templates := "SrcType := USInt" } GE_Contact(in1 := "DL_Vars".Vars.cActualHoursWithoutRunToExerise[1], in2 := "DL_Vars".Vars.cMaxHoursWithoutRunToExerise[1])
      { S7_Templates := "time_type := Time" } "DL_Timer_1_DB".TOF(pt := #tTimeExericePump1, et =>)
      Coil( #xPump1ExeriseRun )
   END_RUNG
   RUNG wire#powerrail
      { S7_Templates := "SrcType := USInt" } GE_Contact(in1 := "DL_Vars".Vars.cActualHoursWithoutRunToExerise[2], in2 := "DL_Vars".Vars.cMaxHoursWithoutRunToExerise[2])
      { S7_Templates := "time_type := Time" } "DL_Timer_2_DB".TOF(pt := #tTimeExericePump2, et =>)
      Coil( #xPump2ExeriseRun )
   END_RUNG
   // the same network as SCL:
   "DL_Timer_1_DB".TOF(IN := "DL_Vars".Vars.cActualHoursWithoutRunToExerise[1] >= "DL_Vars".Vars.cMaxHoursWithoutRunToExerise[1],
                       PT := #tTimeExericePump1);
   #xPump1ExeriseRun := "DL_Timer_1_DB".Q;
   "DL_Timer_2_DB".TOF(IN := "DL_Vars".Vars.cActualHoursWithoutRunToExerise[2] >= "DL_Vars".Vars.cMaxHoursWithoutRunToExerise[2],
                       PT := #tTimeExericePump2);
   #xPump2ExeriseRun := "DL_Timer_2_DB".Q;
END_REGION
END_FUNCTION

FUNCTION "AOProxy" : Void   // FC59001, LAD
{ S7_Optimized_Access := 'TRUE' }
VERSION : 0.1
// stored: AutoNumber false, IsIECCheckEnabled false, SetENOAutomatically false, UDAEnableTagReadback false
   VAR_INPUT
      iUnitID : Int;
      cCHModeCtrl : Byte;
      rDriverSignal : Real;
      rDrivenSignal : Real;
      xProxyIsOnInd : Bool;
      xProxyIsOffInd : Bool;
   END_VAR
   VAR_IN_OUT
      rProxySignal : Real;
      xProxyCmd : Bool;
      xProxyIndError : Bool;
   END_VAR
BEGIN

REGION Network 1 (SCL)
   CASE #cCHModeCtrl OF
       0:  // Not Active
           #xProxyCmd := FALSE;
           #rProxySignal := 0.0;
       1:  // Straignt signal
           #xProxyCmd := TRUE;
           #rProxySignal := #rDrivenSignal;
       2:  // Driven Initial signal
           #xProxyCmd := TRUE;
           #rProxySignal := #rDrivenSignal;
       3:  // Replace initial signal
           #xProxyCmd := TRUE;
           #rProxySignal := #rDriverSignal;
   END_CASE;
END_REGION
END_FUNCTION

FUNCTION "DOProxy" : Void   // FC59002, LAD
{ S7_Optimized_Access := 'TRUE' }
VERSION : 0.1
// stored: AutoNumber false, IsIECCheckEnabled false, SetENOAutomatically false, UDAEnableTagReadback false
   VAR_INPUT
      xInput : Bool;
      xInversion : Bool;   // 0-direct / 1-reverse
      cMOA : Byte;
   END_VAR
   VAR_OUTPUT
      xOutput : Bool;
   END_VAR
   VAR_IN_OUT
      xMemoryOut : Bool;
      xMemoryIn : Bool;
      cMemory : Byte;
      iCounterIn : Int;
      iCounterOut : Int;
   END_VAR
   VAR_TEMP
      InOut_1 : Bool;
   END_VAR
BEGIN

REGION Network 2 (SCL)
   CASE #cMOA OF
       0: // OFF
           #xOutput := FALSE;

       1: // MANUAL
           #xOutput := TRUE;

       2: // AUTO
           #xOutput :=#xInput;

   ELSE
       #xOutput := FALSE;
   END_CASE;
END_REGION

REGION Network 3 (SCL)
   IF #xInversion THEN
       #xOutput := NOT #xOutput;
   END_IF;
END_REGION

REGION Network 4 (SCL)
   IF (#xMemoryIn XOR #xInput) THEN
       IF #iCounterIn > 30000 THEN
           #iCounterIn := 5;
       ELSE
           #iCounterIn := #iCounterIn + 1;
       END_IF;
   END_IF;
   #xMemoryIn := #xInput;
END_REGION

REGION Network 5 (SCL)
   IF (#xMemoryOut XOR #xOutput) THEN
       IF #iCounterOut > 30000 THEN
           #iCounterOut := 5;
       ELSE
           #iCounterOut := #iCounterOut + 1;
       END_IF;
   END_IF;
   #xMemoryOut := #xOutput;
END_REGION
END_FUNCTION

FUNCTION "Proxy_General" : Void   // FC59000, LAD
{ S7_Optimized_Access := 'TRUE' }
VERSION : 0.1
// stored: AutoNumber false, IsIECCheckEnabled false, SetENOAutomatically false, UDAEnableTagReadback false
BEGIN

REGION Network 1
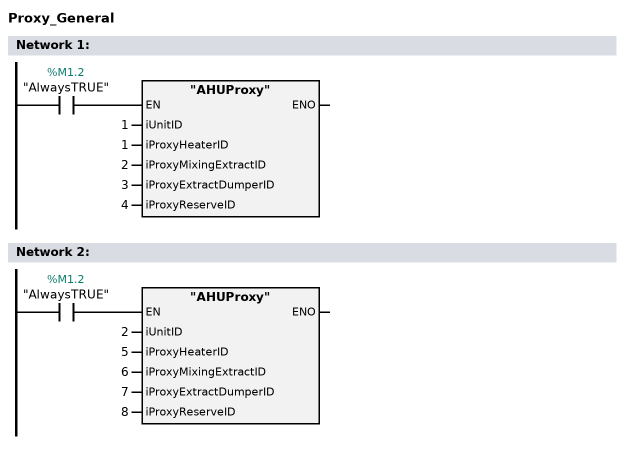
   RUNG wire#powerrail
      Contact( "AlwaysTRUE" )
      "AHUProxy"(iUnitID := 1, iProxyHeaterID := 1, iProxyMixingExtractID := 2, iProxyExtractDumperID := 3, iProxyReserveID := 4)
   END_RUNG
   // the same network as SCL:
   IF "AlwaysTRUE" THEN
       "AHUProxy"(iUnitID := 1,
                  iProxyHeaterID := 1,
                  iProxyMixingExtractID := 2,
                  iProxyExtractDumperID := 3,
                  iProxyReserveID := 4);
   END_IF;
END_REGION

REGION Network 2
   RUNG wire#powerrail
      Contact( "AlwaysTRUE" )
      "AHUProxy"(iUnitID := 2, iProxyHeaterID := 5, iProxyMixingExtractID := 6, iProxyExtractDumperID := 7, iProxyReserveID := 8)
   END_RUNG
   // the same network as SCL:
   IF "AlwaysTRUE" THEN
       "AHUProxy"(iUnitID := 2,
                  iProxyHeaterID := 5,
                  iProxyMixingExtractID := 6,
                  iProxyExtractDumperID := 7,
                  iProxyReserveID := 8);
   END_IF;
END_REGION
END_FUNCTION

FUNCTION "AHUProxy" : Void   // FC59010, LAD
{ S7_Optimized_Access := 'TRUE' }
VERSION : 0.1
// stored: AutoNumber false, IsIECCheckEnabled false, SetENOAutomatically false, UDAEnableTagReadback false
   VAR_INPUT
      iUnitID : Int;   // 1=AHUFood, 2=AHUNonFood
      iProxyHeaterID : Int;
      iProxyMixingExtractID : Int;
      iProxyExtractDumperID : Int;
      iProxyReserveID : Int;
   END_VAR
BEGIN

REGION Network 1: Heater Analog
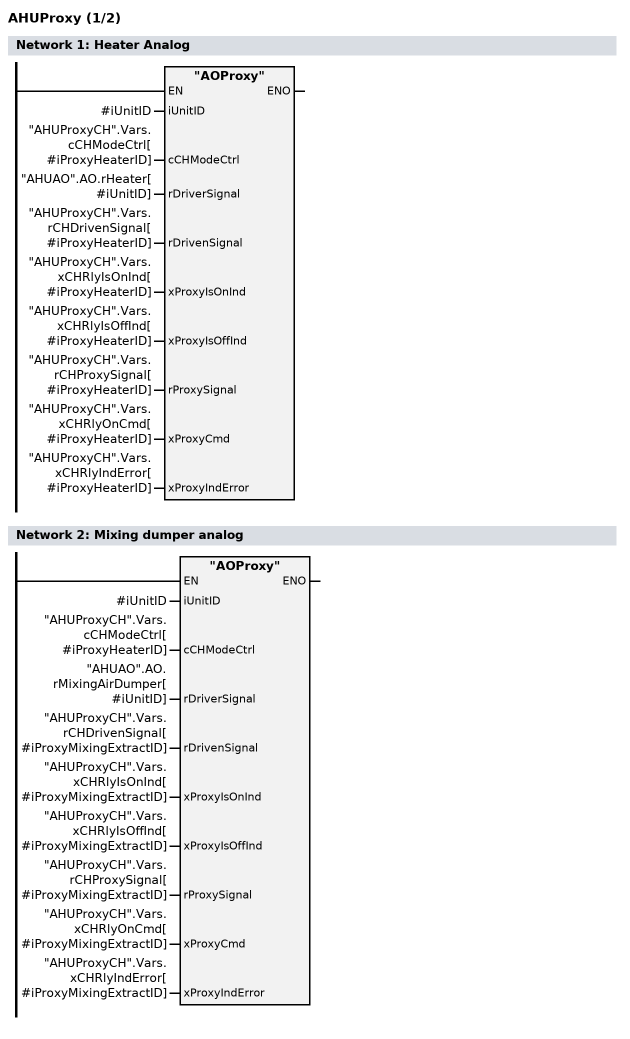
   RUNG wire#powerrail
      "AOProxy"(iUnitID := #iUnitID, cCHModeCtrl := "AHUProxyCH".Vars.cCHModeCtrl[#iProxyHeaterID], rDriverSignal := "AHUAO".AO.rHeater[#iUnitID], rDrivenSignal := "AHUProxyCH".Vars.rCHDrivenSignal[#iProxyHeaterID], xProxyIsOnInd := "AHUProxyCH".Vars.xCHRlyIsOnInd[#iProxyHeaterID], xProxyIsOffInd := "AHUProxyCH".Vars.xCHRlyIsOffInd[#iProxyHeaterID], rProxySignal := "AHUProxyCH".Vars.rCHProxySignal[#iProxyHeaterID], xProxyCmd := "AHUProxyCH".Vars.xCHRlyOnCmd[#iProxyHeaterID], xProxyIndError := "AHUProxyCH".Vars.xCHRlyIndError[#iProxyHeaterID])
   END_RUNG
   // the same network as SCL:
   "AOProxy"(iUnitID := #iUnitID,
             cCHModeCtrl := "AHUProxyCH".Vars.cCHModeCtrl[#iProxyHeaterID],
             rDriverSignal := "AHUAO".AO.rHeater[#iUnitID],
             rDrivenSignal := "AHUProxyCH".Vars.rCHDrivenSignal[#iProxyHeaterID],
             xProxyIsOnInd := "AHUProxyCH".Vars.xCHRlyIsOnInd[#iProxyHeaterID],
             xProxyIsOffInd := "AHUProxyCH".Vars.xCHRlyIsOffInd[#iProxyHeaterID],
             rProxySignal := "AHUProxyCH".Vars.rCHProxySignal[#iProxyHeaterID],
             xProxyCmd := "AHUProxyCH".Vars.xCHRlyOnCmd[#iProxyHeaterID],
             xProxyIndError := "AHUProxyCH".Vars.xCHRlyIndError[#iProxyHeaterID]);
END_REGION

REGION Network 2: Mixing dumper analog
   RUNG wire#powerrail
      "AOProxy"(iUnitID := #iUnitID, cCHModeCtrl := "AHUProxyCH".Vars.cCHModeCtrl[#iProxyHeaterID], rDriverSignal := "AHUAO".AO.rMixingAirDumper[#iUnitID], rDrivenSignal := "AHUProxyCH".Vars.rCHDrivenSignal[#iProxyMixingExtractID], xProxyIsOnInd := "AHUProxyCH".Vars.xCHRlyIsOnInd[#iProxyMixingExtractID], xProxyIsOffInd := "AHUProxyCH".Vars.xCHRlyIsOffInd[#iProxyMixingExtractID], rProxySignal := "AHUProxyCH".Vars.rCHProxySignal[#iProxyMixingExtractID], xProxyCmd := "AHUProxyCH".Vars.xCHRlyOnCmd[#iProxyMixingExtractID], xProxyIndError := "AHUProxyCH".Vars.xCHRlyIndError[#iProxyMixingExtractID])
   END_RUNG
   // the same network as SCL:
   "AOProxy"(iUnitID := #iUnitID,
             cCHModeCtrl := "AHUProxyCH".Vars.cCHModeCtrl[#iProxyHeaterID],
             rDriverSignal := "AHUAO".AO.rMixingAirDumper[#iUnitID],
             rDrivenSignal := "AHUProxyCH".Vars.rCHDrivenSignal[#iProxyMixingExtractID],
             xProxyIsOnInd := "AHUProxyCH".Vars.xCHRlyIsOnInd[#iProxyMixingExtractID],
             xProxyIsOffInd := "AHUProxyCH".Vars.xCHRlyIsOffInd[#iProxyMixingExtractID],
             rProxySignal := "AHUProxyCH".Vars.rCHProxySignal[#iProxyMixingExtractID],
             xProxyCmd := "AHUProxyCH".Vars.xCHRlyOnCmd[#iProxyMixingExtractID],
             xProxyIndError := "AHUProxyCH".Vars.xCHRlyIndError[#iProxyMixingExtractID]);
END_REGION

REGION Network 3: Mixing dumper analog
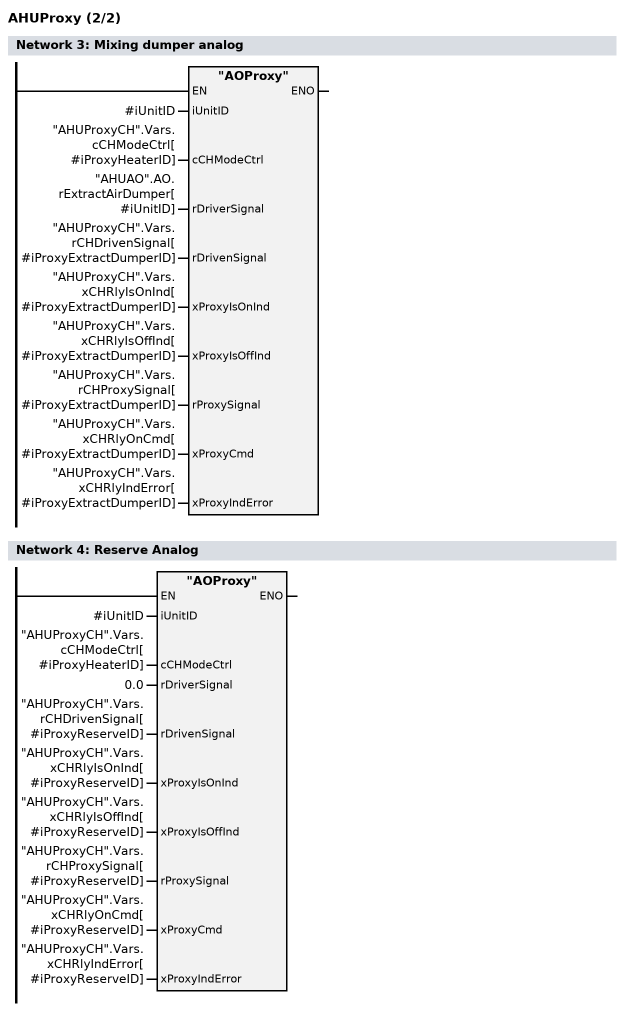
   RUNG wire#powerrail
      "AOProxy"(iUnitID := #iUnitID, cCHModeCtrl := "AHUProxyCH".Vars.cCHModeCtrl[#iProxyHeaterID], rDriverSignal := "AHUAO".AO.rExtractAirDumper[#iUnitID], rDrivenSignal := "AHUProxyCH".Vars.rCHDrivenSignal[#iProxyExtractDumperID], xProxyIsOnInd := "AHUProxyCH".Vars.xCHRlyIsOnInd[#iProxyExtractDumperID], xProxyIsOffInd := "AHUProxyCH".Vars.xCHRlyIsOffInd[#iProxyExtractDumperID], rProxySignal := "AHUProxyCH".Vars.rCHProxySignal[#iProxyExtractDumperID], xProxyCmd := "AHUProxyCH".Vars.xCHRlyOnCmd[#iProxyExtractDumperID], xProxyIndError := "AHUProxyCH".Vars.xCHRlyIndError[#iProxyExtractDumperID])
   END_RUNG
   // the same network as SCL:
   "AOProxy"(iUnitID := #iUnitID,
             cCHModeCtrl := "AHUProxyCH".Vars.cCHModeCtrl[#iProxyHeaterID],
             rDriverSignal := "AHUAO".AO.rExtractAirDumper[#iUnitID],
             rDrivenSignal := "AHUProxyCH".Vars.rCHDrivenSignal[#iProxyExtractDumperID],
             xProxyIsOnInd := "AHUProxyCH".Vars.xCHRlyIsOnInd[#iProxyExtractDumperID],
             xProxyIsOffInd := "AHUProxyCH".Vars.xCHRlyIsOffInd[#iProxyExtractDumperID],
             rProxySignal := "AHUProxyCH".Vars.rCHProxySignal[#iProxyExtractDumperID],
             xProxyCmd := "AHUProxyCH".Vars.xCHRlyOnCmd[#iProxyExtractDumperID],
             xProxyIndError := "AHUProxyCH".Vars.xCHRlyIndError[#iProxyExtractDumperID]);
END_REGION

REGION Network 4: Reserve Analog
   RUNG wire#powerrail
      "AOProxy"(iUnitID := #iUnitID, cCHModeCtrl := "AHUProxyCH".Vars.cCHModeCtrl[#iProxyHeaterID], rDriverSignal := 0.0, rDrivenSignal := "AHUProxyCH".Vars.rCHDrivenSignal[#iProxyReserveID], xProxyIsOnInd := "AHUProxyCH".Vars.xCHRlyIsOnInd[#iProxyReserveID], xProxyIsOffInd := "AHUProxyCH".Vars.xCHRlyIsOffInd[#iProxyReserveID], rProxySignal := "AHUProxyCH".Vars.rCHProxySignal[#iProxyReserveID], xProxyCmd := "AHUProxyCH".Vars.xCHRlyOnCmd[#iProxyReserveID], xProxyIndError := "AHUProxyCH".Vars.xCHRlyIndError[#iProxyReserveID])
   END_RUNG
   // the same network as SCL:
   "AOProxy"(iUnitID := #iUnitID,
             cCHModeCtrl := "AHUProxyCH".Vars.cCHModeCtrl[#iProxyHeaterID],
             rDriverSignal := 0.0,
             rDrivenSignal := "AHUProxyCH".Vars.rCHDrivenSignal[#iProxyReserveID],
             xProxyIsOnInd := "AHUProxyCH".Vars.xCHRlyIsOnInd[#iProxyReserveID],
             xProxyIsOffInd := "AHUProxyCH".Vars.xCHRlyIsOffInd[#iProxyReserveID],
             rProxySignal := "AHUProxyCH".Vars.rCHProxySignal[#iProxyReserveID],
             xProxyCmd := "AHUProxyCH".Vars.xCHRlyOnCmd[#iProxyReserveID],
             xProxyIndError := "AHUProxyCH".Vars.xCHRlyIndError[#iProxyReserveID]);
END_REGION
END_FUNCTION

FUNCTION "AObasic" : Void   // FC10002, FBD
{ S7_Optimized_Access := 'TRUE' }
VERSION : 0.1
// stored: AutoNumber false, IsIECCheckEnabled false, SetENOAutomatically false, UDAEnableTagReadback false
   VAR_INPUT
      rInput : Real;   // 0 to 100
      cM0A : Byte;   // 0-direct / 1-reverse / 0-outp_off / 1- out=MAN_OUTPUT /2 -out=input
      rManOutput : Real;
   END_VAR
   VAR_OUTPUT
      iOutput : Int;
   END_VAR
   VAR_TEMP
      rOut : Real;
      iOut : Int;
      rManOutputTemp : Real;
      iManOutputTemp : Int;
   END_VAR
BEGIN

REGION Network 1
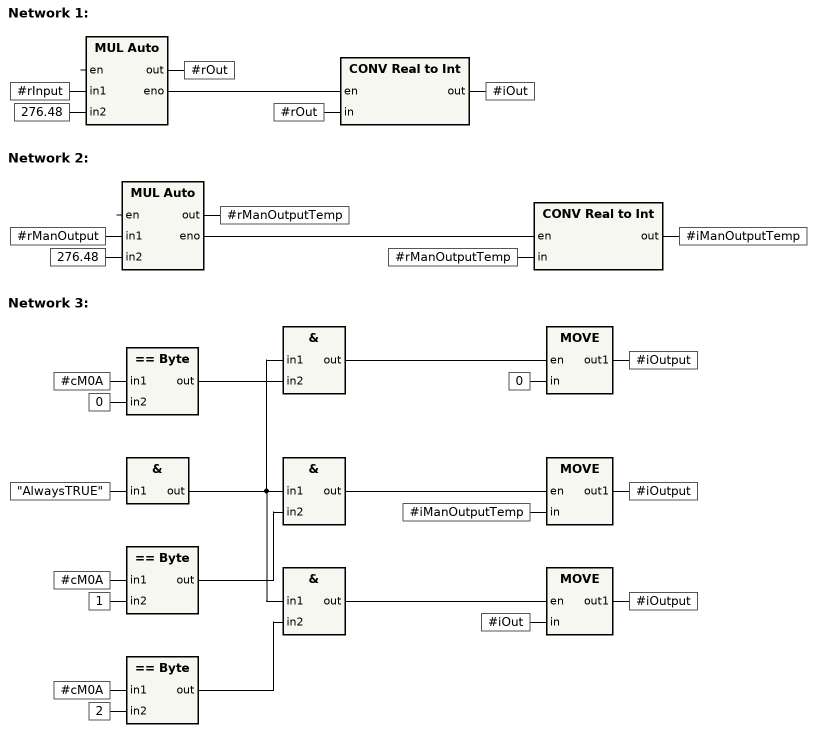
   #rOut := #rInput * 276.48;
   #iOut := REAL_TO_INT(#rOut);
END_REGION

REGION Network 2
   #rManOutputTemp := #rManOutput * 276.48;
   #iManOutputTemp := REAL_TO_INT(#rManOutputTemp);
END_REGION

REGION Network 3
   IF "AlwaysTRUE" AND (#cM0A = 0) THEN #iOutput := 0; END_IF;
   IF "AlwaysTRUE" AND (#cM0A = 1) THEN #iOutput := #iManOutputTemp; END_IF;
   IF "AlwaysTRUE" AND (#cM0A = 2) THEN #iOutput := #iOut; END_IF;
END_REGION
END_FUNCTION

FUNCTION "DIbasic" : Void   // FC10003, LAD
{ S7_Optimized_Access := 'TRUE' }
VERSION : 0.1
// stored: AutoNumber false, IsIECCheckEnabled false, SetENOAutomatically false, UDAEnableTagReadback false
   VAR_INPUT
      xInput : Bool;
      xInversion : Bool;   // 0-direct / 1-reverse
   END_VAR
   VAR_OUTPUT
      xOutputFiltered : Bool;
   END_VAR
   VAR_IN_OUT
      iAddImpOff : Int;
      xMemory : Bool;
      iAddImpOn : Int;
      iCounter : Int;
   END_VAR
   VAR_TEMP
      InOut_1 : Bool;
   END_VAR
   VAR_TEMP   // added for the SCL form of the ladder/FBD networks
      _w1 : Bool;
      _w2 : Bool;
   END_VAR
BEGIN

REGION Network 1 (FBD)
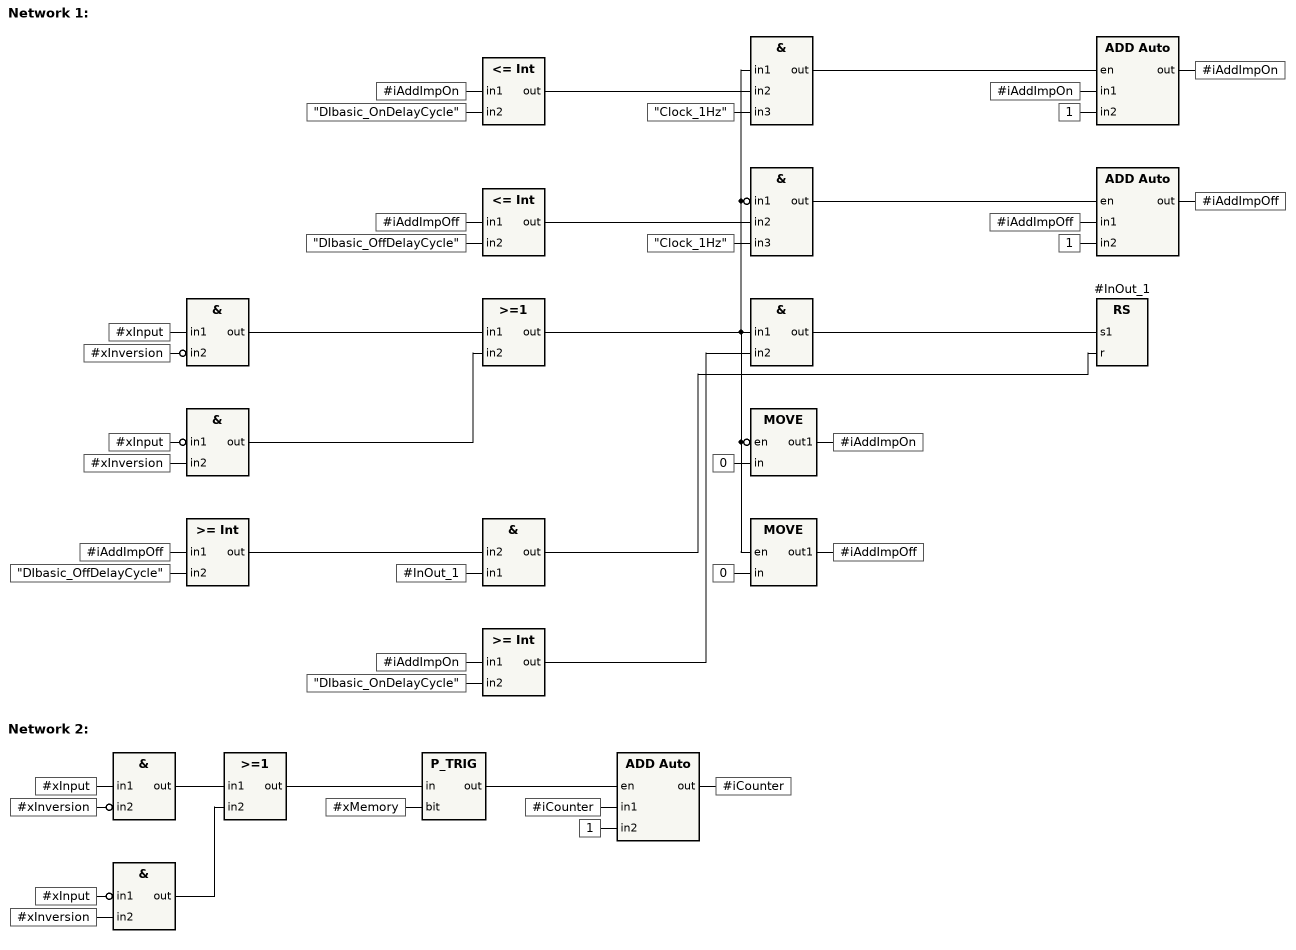
   #_w1 := (#xInput AND NOT #xInversion) OR (NOT #xInput AND #xInversion);
   IF #_w1 AND (#iAddImpOn <= "DIbasic_OnDelayCycle") AND "Clock_1Hz" THEN
       #iAddImpOn := #iAddImpOn + 1;
   END_IF;
   IF NOT #_w1 AND (#iAddImpOff <= "DIbasic_OffDelayCycle") AND "Clock_1Hz" THEN
       #iAddImpOff := #iAddImpOff + 1;
   END_IF;
   IF (#iAddImpOff >= "DIbasic_OffDelayCycle") AND #InOut_1 THEN
       #InOut_1 := FALSE;   // RS flip-flop
   END_IF;
   IF #_w1 AND (#iAddImpOn >= "DIbasic_OnDelayCycle") THEN #InOut_1 := TRUE; END_IF;
   IF NOT #_w1 THEN #iAddImpOn := 0; END_IF;
   IF #_w1 THEN #iAddImpOff := 0; END_IF;
END_REGION

REGION Network 2 (FBD)
   #_w1 := (#xInput AND NOT #xInversion) OR (NOT #xInput AND #xInversion);
   #_w2 := #_w1 AND NOT #xMemory;   // rising edge
   #xMemory := #_w1;
   IF #_w2 THEN #iCounter := #iCounter + 1; END_IF;
END_REGION

REGION Network 3
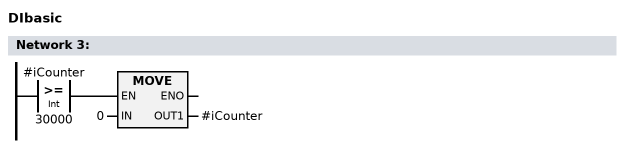
   RUNG wire#powerrail
      { S7_Templates := "SrcType := Int" } GE_Contact(in1 := #iCounter, in2 := 30000)
      Move(in := 0, out1 => #iCounter)
   END_RUNG
   // the same network as SCL:
   IF #iCounter >= 30000 THEN #iCounter := 0; END_IF;
END_REGION
END_FUNCTION

FUNCTION "DObasic" : Void   // FC10004, FBD
{ S7_Optimized_Access := 'TRUE' }
VERSION : 0.1
// stored: AutoNumber false, IsIECCheckEnabled false, SetENOAutomatically false, UDAEnableTagReadback false
   VAR_INPUT
      xInput : Bool;
      cM0A : Byte;   // 0-direct / 1-reverse / 0-outp_off / 1- aut=1 /2 -out=input
   END_VAR
   VAR_OUTPUT
      iCounter : Int;
      xOutput : Bool;
   END_VAR
   VAR_IN_OUT
      Bit_Count_1 : Bool;
   END_VAR
   VAR_TEMP
      cM0A_0 : Bool;
      cM0A_1 : Bool;
      cM0A_2 : Bool;
   END_VAR
   VAR CONSTANT
      bit_count : Bool;
   END_VAR
   VAR_TEMP   // added for the SCL form of the ladder/FBD networks
      _w1 : Bool;
   END_VAR
BEGIN

REGION Network 1
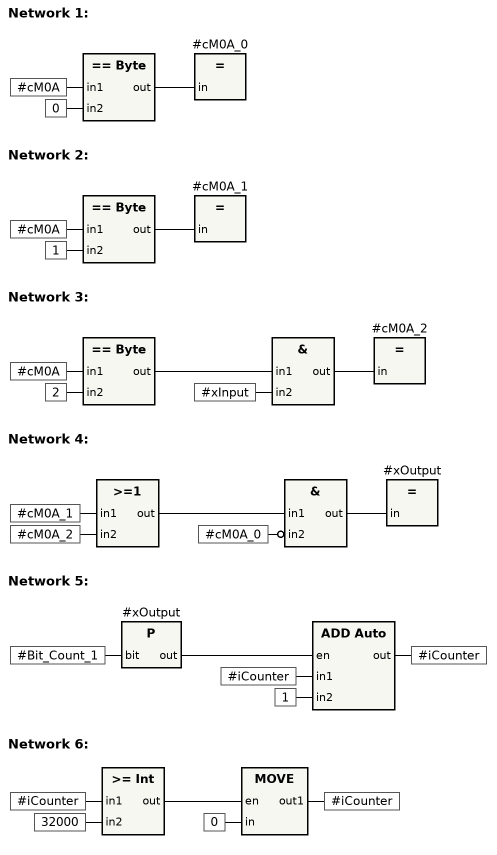
   #cM0A_0 := #cM0A = 0;
END_REGION

REGION Network 2
   #cM0A_1 := #cM0A = 1;
END_REGION

REGION Network 3
   #cM0A_2 := (#cM0A = 2) AND #xInput;
END_REGION

REGION Network 4
   #xOutput := (#cM0A_1 OR #cM0A_2) AND NOT #cM0A_0;
END_REGION

REGION Network 5
   #_w1 := #xOutput AND NOT #Bit_Count_1;   // rising edge of #xOutput
   #Bit_Count_1 := #xOutput;
   IF #_w1 THEN #iCounter := #iCounter + 1; END_IF;
END_REGION

REGION Network 6
   IF #iCounter >= 32000 THEN #iCounter := 0; END_IF;
END_REGION
END_FUNCTION

FUNCTION "BoilerActualUnitStatesCtrl" : Void   // FC60108, LAD
{ S7_Optimized_Access := 'TRUE' }
VERSION : 0.1
// Operation Modes                                                 Unit State
// 0=Protection                                                         0=Stopped
// 1=Economy                                                           1=Checking-up  
// 2=PreComfort                                                       2=Preheating
// 3=Comfor                                                              3=Starting 
// 4=Auto(Scheduler)                                              4=RecirculatingOperation
//                                                                                 5=Economy Operation                                                                                                                                            6=PreComfort Operation 
//                                                                                 7=Comfort  operation
//                                                                                 8=Stopping
//                                                                                 9 =Blocking
// stored: AutoNumber false, IsIECCheckEnabled false, SetENOAutomatically false, UDAEnableTagReadback false
   VAR_INPUT
      iUnitID : Int;
      xManualSummer : Bool;
      xManualWinter : Bool;
      cTargetUnitState : Byte;
      cFromHotToColdDelay : Byte;
   END_VAR
   VAR_OUTPUT
      iUnitStateForHMI : Int;
   END_VAR
   VAR_IN_OUT
      cNextUnitState : Byte;
   END_VAR
   VAR_TEMP
      cState : Byte;
   END_VAR
BEGIN

REGION Network 1 (SCL)
   (*
   "BoilerUnitStates".UnitStates.cActual[#iUnitID] = UnitStates.cTarget[iUnitID];
   *)
END_REGION

REGION Network 2 (SCL): Simple state for HMI
END_REGION
END_FUNCTION

FUNCTION "BoilerModesCtrlAutoMode" : Void   // FC60106, LAD
{ S7_Optimized_Access := 'TRUE' }
VERSION : 0.1
// stored: AutoNumber false, IsIECCheckEnabled false, SetENOAutomatically false, UDAEnableTagReadback false
   VAR_INPUT
      cPreselectedPLCOpMode : Byte;
      cSchedulerTargetOpMode : Byte;
      cPanelSelectorActualMode : Byte;
   END_VAR
   VAR_OUTPUT
      cTargetOpMode : Byte;
      cActualOpMode : Byte;
   END_VAR
   VAR_TEMP
      TargetUnitMode_old : Int;
      ResetActualOperationMode : Bool;
   END_VAR
BEGIN

REGION Network 1 (SCL)
   CASE #cPanelSelectorActualMode OF
       0:                                                     // Switch is in Summer/OFF
           #cTargetOpMode := 0;                               //Summer
       1:                                                     // ON
           #cTargetOpMode := 1;                               // Winter 
       ELSE                                                   // Switch is in Auto
           IF #cPreselectedPLCOpMode = 2 THEN                 // PLC mode 2=Scheduler
               #cTargetOpMode := #cSchedulerTargetOpMode;     // 
           ELSE                                               //mode-0-1-2-
               #cTargetOpMode := #cPreselectedPLCOpMode;
           END_IF;
   END_CASE;
END_REGION

REGION Network 2 (SCL)
   IF #cTargetOpMode <> #cActualOpMode THEN
       // Update Actual OP Mode
       #cActualOpMode := #cTargetOpMode;
   END_IF;
END_REGION

REGION Network 3 (SCL)
   IF #cActualOpMode <> "cActualOpModePrevOne" THEN
       "iActualOpModeCounter" := "iActualOpModeCounter" + 1;
   END_IF;
END_REGION
END_FUNCTION

FUNCTION "Boiler_TargetUnitStatesCtrl" : Void   // FC60107, LAD
{ S7_Optimized_Access := 'TRUE' }
VERSION : 0.1
// Operation Modes                                                 Unit State
// 0=Protection                                                         0=Stopped
// 1=Economy                                                           1=Checking-up  
// 2=PreComfort                                                       2=Preheating
// 3=Comfor                                                              3=Starting 
// 4=Auto(Scheduler)                                              4=RecirculatingOperation
//                                                                                 5=Economy Operation                                                                                                                                            6=PreComfort Operation 
//                                                                                 7=Comfort  operation
//                                                                                 8=Stopping
//                                                                                 9=Blocking
// stored: AutoNumber false, IsIECCheckEnabled false, SetENOAutomatically false, UDAEnableTagReadback false
   VAR_INPUT
      cActualOpMode : Byte;
      xHeatingActiveByOATRequest : Bool;
      xHeatingActiveBySecondBoilerAlarm : Bool;
      xBlockByAlarm : Bool;
      xIsReady : Bool;
   END_VAR
   VAR_OUTPUT
      cTargetUnitState : Byte;
      xRequestBackupToAnotherBoiler : Bool;
   END_VAR
BEGIN

REGION Network 1 (SCL)
   CASE #cActualOpMode OF
       0:                                                  // OpMode is OFF(Protection)
           IF #xBlockByAlarm THEN                               // Stop by alarm      
               #cTargetUnitState := 9;
           ELSE 
               #cTargetUnitState := 0;
           END_IF;
       1:                                                  // Economy mode 
           IF #xBlockByAlarm THEN                               // Stop by alarm      
               #cTargetUnitState := 9;
           ELSIF #xHeatingActiveByOATRequest THEN                           //Time to start
               #cTargetUnitState := 5;
           ELSE                                                // Stop by no request
               #cTargetUnitState := 0;
           END_IF;
       2:                                                  // PreComfort mode 
           IF #xBlockByAlarm THEN                               // Stop by alarm      
               #cTargetUnitState := 9;
           ELSIF #xHeatingActiveByOATRequest THEN                           //Time to start
               #cTargetUnitState := 6;
           ELSE                                                // Stop by no request
               #cTargetUnitState := 0;
           END_IF;
       3:                                                      // Comfort mode 
           IF #xBlockByAlarm THEN                               // Stop by alarm      
               #cTargetUnitState := 9;
           ELSIF #xHeatingActiveByOATRequest THEN                           //Time to start
               #cTargetUnitState := 7;
           ELSE                                                // Stop by no request
               #cTargetUnitState := 0;
           END_IF;
       ELSE:
           IF #xBlockByAlarm THEN                               // Stop by alarm      
               #cTargetUnitState := 9;
           ELSE
               #cTargetUnitState := 0;
           END_IF;
   END_CASE;
END_REGION

REGION Network 2 (SCL)
   IF #cTargetUnitState <> "cTargetUnitStatePrevOne" THEN
       "iTargetUnitStareCounter" := "iTargetUnitStareCounter" + 1;
   END_IF;

   "cTargetUnitStatePrevOne" := #cTargetUnitState;
END_REGION
END_FUNCTION

FUNCTION "Boiler_UnitState" : Void   // FC61000, FBD
{ S7_Optimized_Access := 'TRUE' }
VERSION : 0.1
// BoilerOpMode                                        BoilerUnitState
// 0-OFF/Summer                                       0 Off
// 1-On/Winter                                             1 ColdStandBy
//                                                                   1 HotStandBy
//                                                                   2 Heating
// stored: AutoNumber false, IsIECCheckEnabled false, SetENOAutomatically false, UDAEnableTagReadback false
   VAR_INPUT
      rOAT : Real;
      rBoiler1OATOff : Real;
      rBoiler1OATOn : Real;
      rBoiler2OAT1On : Real;
      rBoiler2OAT1Off : Real;
      rBoiler2OAT2On : Real;
      rBoiler2OAT2Off : Real;
   END_VAR
   VAR_IN_OUT
      xBoiler1OATRequest : Bool;
      xBoiler2OATRequest : Bool;
   END_VAR
   VAR_TEMP
      FA_temp : Real;
      xB1State : Bool;
      xB2Band1State : Bool;
      xB2Band2State : Bool;
      xB2Band1Effective : Bool;
   END_VAR
BEGIN

REGION Network 1 (SCL)
   IF "FirstScan" THEN
       ;
       //"AHUUnitStates".UnitStates.cActual[#iUnitID] := 0;
       //"AHUUnitStates".UnitStates.cTarget[#iUnitID] := 0;
   END_IF;
END_REGION

REGION Network 2 (SCL): Boiler1 Select from Panel
   IF "HSsDI".Requests.xSeasonAuto[1] THEN
       "BoilerOpModes".OpModes.cPreselectedOpModePanel[1] := 2;//Auto
   ELSIF "HSsDI".Requests.xSeasonWinter[1] THEN
       "BoilerOpModes".OpModes.cPreselectedOpModePanel[1]:= 1;//Winter - Always On
   ELSE
       "BoilerOpModes".OpModes.cPreselectedOpModePanel[1] := 0;//Summer - Off
   END_IF;
END_REGION

REGION Network 3 (SCL): Boiler2 Select from Panel
   IF "BoilerOpModes".OpModes.xBoiler2IndividualPanelSwitch THEN
       IF "HSsDI".Requests.xSeasonAuto[2] THEN
           "BoilerOpModes".OpModes.cPreselectedOpModePanel[2] := 2;//Auto
       ELSIF "HSsDI".Requests.xSeasonWinter[2] THEN
           "BoilerOpModes".OpModes.cPreselectedOpModePanel[2] := 1;//Winter - Always On
       ELSE
           "BoilerOpModes".OpModes.cPreselectedOpModePanel[2] := 0;//Summer - Off
       END_IF;
   ELSE
       IF "HSsDI".Requests.xSeasonAuto[1] THEN
           "BoilerOpModes".OpModes.cPreselectedOpModePanel[2] := 2;//Auto
       ELSIF "HSsDI".Requests.xSeasonWinter[1] THEN
           "BoilerOpModes".OpModes.cPreselectedOpModePanel[2] := 1;//Winter - Always On
       ELSE
           "BoilerOpModes".OpModes.cPreselectedOpModePanel[2] := 0;//Summer - Off
       END_IF;
   END_IF;
END_REGION

REGION Network 4: Boiler1 Actual Operation Mode define
   // Operation Modes                                                 Unit State
   // 0=Protection                                                         0=Stopped
   // 1=Economy                                                           1=Checking-up  
   // 2=PreComfort                                                       2=Preheating
   // 3=Comfor                                                              3=Starting 
   // 4=Auto(Scheduler)                                              4=RecirculatingOperation (Protection)
   //                                                                                 5=Sustained Mode (Economy setpoints)
   //                                                                                 6=Sustained Mode (PreComfort setpoints) 
   //                                                                                 7=Comfort  operation
   //                                                                                 8=Stopping
   //                                                                                 9=Blocking
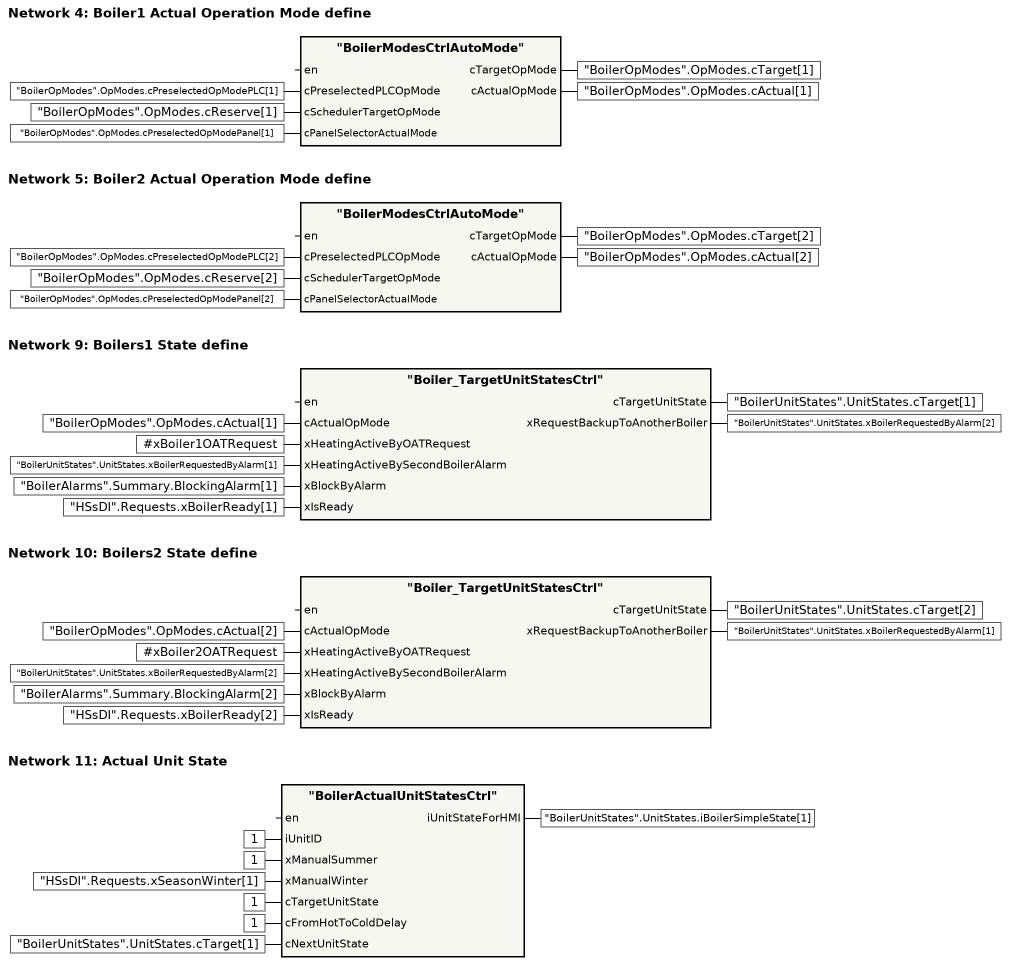
   "BoilerModesCtrlAutoMode"(cPreselectedPLCOpMode := "BoilerOpModes".OpModes.cPreselectedOpModePLC[1],
                           cSchedulerTargetOpMode := "BoilerOpModes".OpModes.cReserve[1],
                           cPanelSelectorActualMode := "BoilerOpModes".OpModes.cPreselectedOpModePanel[1],
                           cTargetOpMode => "BoilerOpModes".OpModes.cTarget[1],
                           cActualOpMode => "BoilerOpModes".OpModes.cActual[1]);
END_REGION

REGION Network 5: Boiler2 Actual Operation Mode define
   "BoilerModesCtrlAutoMode"(cPreselectedPLCOpMode := "BoilerOpModes".OpModes.cPreselectedOpModePLC[2],
                           cSchedulerTargetOpMode := "BoilerOpModes".OpModes.cReserve[2],
                           cPanelSelectorActualMode := "BoilerOpModes".OpModes.cPreselectedOpModePanel[2],
                           cTargetOpMode => "BoilerOpModes".OpModes.cTarget[2],
                           cActualOpMode => "BoilerOpModes".OpModes.cActual[2]);
END_REGION

REGION Network 6 (SCL): Boiler1 request by OAT
   IF NOT #xB1State THEN
       // Вмикаємо котел 1, коли стало достатньо холодно
       IF #rOAT <= #rBoiler1OATOn THEN
           #xB1State := TRUE;
       END_IF;
   ELSE
       // Вимикаємо котел 1, коли потеплішало вище абсолютного порогу
       IF #rOAT >= #rBoiler1OATOff THEN
           #xB1State := FALSE;
       END_IF;
   END_IF;

   #xBoiler1OATRequest := #xB1State;
END_REGION

REGION Network 7 (SCL): Boiler2 request by OAT, OAT range 1
   // Помірний холод»Помірний холод»: дозволяти лише доти, доки котел 1 ще НЕ увімкнувся.
   // // Пороги незалежні й реалізовані абсолютними значеннями
   IF NOT #xB2Band1State THEN
       IF #rOAT <= #rBoiler2OAT1On THEN
           #xB2Band1State := TRUE;
       END_IF;
   ELSE
       IF #rOAT >= #rBoiler2OAT1Off THEN
           #xB2Band1State := FALSE;
       END_IF;
   END_IF;

   // Маскуємо Band1, якщо котел 1 вже дозволений (умова "до включення першого котла")
   #xB2Band1Effective := #xB2Band1State AND (NOT #xBoiler1OATRequest);
END_REGION

REGION Network 8 (SCL): Boiler2 request by OAT, OAT range 2
   // «Сильний мороз»: дозволяти незалежно від стану котла 1.
   IF NOT #xB2Band2State THEN
       IF #rOAT <= #rBoiler2OAT2On THEN
           #xB2Band2State := TRUE;
       END_IF;
   ELSE
       IF #rOAT >= #rBoiler2OAT2Off THEN
           #xB2Band2State := FALSE;
       END_IF;
   END_IF;

   #xBoiler2OATRequest := #xB2Band2State OR #xB2Band1Effective;
END_REGION

REGION Network 9: Boilers1 State define
   // Operation Modes                                                 Unit State
   "Boiler_TargetUnitStatesCtrl"(cActualOpMode := "BoilerOpModes".OpModes.cActual[1],
                           xHeatingActiveByOATRequest := #xBoiler1OATRequest,
                           xHeatingActiveBySecondBoilerAlarm := "BoilerUnitStates".UnitStates.xBoilerRequestedByAlarm[1],
                           xBlockByAlarm := "BoilerAlarms".Summary.BlockingAlarm[1],
                           xIsReady := "HSsDI".Requests.xBoilerReady[1],
                           cTargetUnitState => "BoilerUnitStates".UnitStates.cTarget[1],
                           xRequestBackupToAnotherBoiler => "BoilerUnitStates".UnitStates.xBoilerRequestedByAlarm[2]);
END_REGION

REGION Network 10: Boilers2 State define
   // Operation Modes                                                 Unit State
   "Boiler_TargetUnitStatesCtrl"(cActualOpMode := "BoilerOpModes".OpModes.cActual[2],
                           xHeatingActiveByOATRequest := #xBoiler2OATRequest,
                           xHeatingActiveBySecondBoilerAlarm := "BoilerUnitStates".UnitStates.xBoilerRequestedByAlarm[2],
                           xBlockByAlarm := "BoilerAlarms".Summary.BlockingAlarm[2],
                           xIsReady := "HSsDI".Requests.xBoilerReady[2],
                           cTargetUnitState => "BoilerUnitStates".UnitStates.cTarget[2],
                           xRequestBackupToAnotherBoiler => "BoilerUnitStates".UnitStates.xBoilerRequestedByAlarm[1]);
END_REGION

REGION Network 11: Actual Unit State
   "BoilerActualUnitStatesCtrl"(iUnitID := 1,
                           xManualSummer := 1,
                           xManualWinter := "HSsDI".Requests.xSeasonWinter[1],
                           cTargetUnitState := 1,
                           cFromHotToColdDelay := 1,
                           cNextUnitState := "BoilerUnitStates".UnitStates.cTarget[1],
                           iUnitStateForHMI => "BoilerUnitStates".UnitStates.iBoilerSimpleState[1]);
END_REGION
END_FUNCTION

FUNCTION "Boiler_Main" : Void   // FC1010, LAD
{ S7_Optimized_Access := 'TRUE' }
VERSION : 0.1
// stored: AutoNumber false, IsIECCheckEnabled false, SetENOAutomatically false, UDAEnableTagReadback false
BEGIN

REGION Network 1
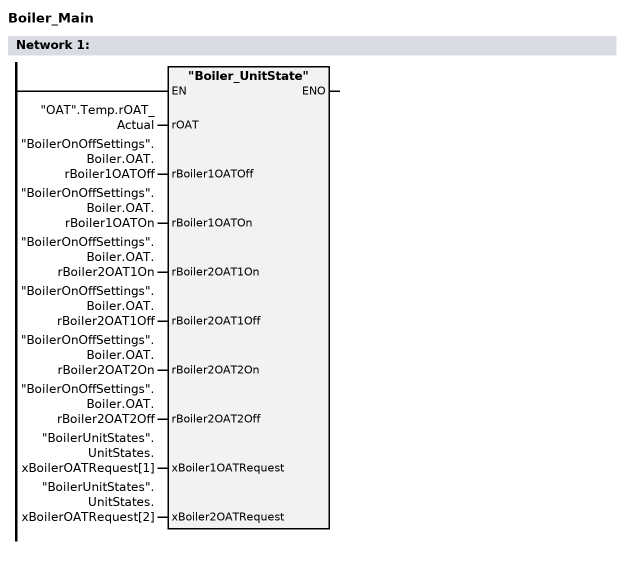
   RUNG wire#powerrail
      "Boiler_UnitState"(rOAT := "OAT".Temp.rOAT_Actual, rBoiler1OATOff := "BoilerOnOffSettings".Boiler.OAT.rBoiler1OATOff, rBoiler1OATOn := "BoilerOnOffSettings".Boiler.OAT.rBoiler1OATOn, rBoiler2OAT1On := "BoilerOnOffSettings".Boiler.OAT.rBoiler2OAT1On, rBoiler2OAT1Off := "BoilerOnOffSettings".Boiler.OAT.rBoiler2OAT1Off, rBoiler2OAT2On := "BoilerOnOffSettings".Boiler.OAT.rBoiler2OAT2On, rBoiler2OAT2Off := "BoilerOnOffSettings".Boiler.OAT.rBoiler2OAT2Off, xBoiler1OATRequest := "BoilerUnitStates".UnitStates.xBoilerOATRequest[1], xBoiler2OATRequest := "BoilerUnitStates".UnitStates.xBoilerOATRequest[2])
   END_RUNG
   // the same network as SCL:
   "Boiler_UnitState"(rOAT := "OAT".Temp.rOAT_Actual,
                      rBoiler1OATOff := "BoilerOnOffSettings".Boiler.OAT.rBoiler1OATOff,
                      rBoiler1OATOn := "BoilerOnOffSettings".Boiler.OAT.rBoiler1OATOn,
                      rBoiler2OAT1On := "BoilerOnOffSettings".Boiler.OAT.rBoiler2OAT1On,
                      rBoiler2OAT1Off := "BoilerOnOffSettings".Boiler.OAT.rBoiler2OAT1Off,
                      rBoiler2OAT2On := "BoilerOnOffSettings".Boiler.OAT.rBoiler2OAT2On,
                      rBoiler2OAT2Off := "BoilerOnOffSettings".Boiler.OAT.rBoiler2OAT2Off,
                      xBoiler1OATRequest := "BoilerUnitStates".UnitStates.xBoilerOATRequest[1],
                      xBoiler2OATRequest := "BoilerUnitStates".UnitStates.xBoilerOATRequest[2]);
END_REGION
END_FUNCTION

FUNCTION "AHURegsAndTargetStatesInComfortOpMode" : Void   // FC60033, LAD
{ S7_Optimized_Access := 'TRUE' }
VERSION : 0.1
// Operation Modes                                                 Unit State
// 0=                                                                            0=Stopped
// 1                                                                              1=Checking-up  
// 2                                                                              2=Preheating
// 3 = Comfort                                                           3=Starting 
//                                                                                 4=RecirculatingOperation (Protection)
//                                                                                 Not 5=Sustained Mode (Economy)
//                                                                                 Not 6=Sustained Mode (PreComfort setpoints) 
//                                                                                 7=Comfort  operation
//                                                                                 Not 8=Night Cooling
//                                                                                 9=Stopping
//                                                                                 10=Blocking
//                                                                                 11=FrostProtecting
// stored: AutoNumber false, IsIECCheckEnabled false, SetENOAutomatically false, UDAEnableTagReadback false
   VAR_INPUT
      iUnitID : Int;
      cActualOpMode : Byte;
      cHeatingRegCfg : Byte;
      cCoolingRegCfg : Byte;
      cIAQRegCfg : Byte;
      cBuildingdPRegCfg : Byte;
   END_VAR
   VAR_OUTPUT
      cTargetState : Byte;
      cHeatingRegState : Byte;
      cCoolingRegState : Byte;
      cIAQRegState : Byte;
      cBuildingdPRegState : Byte;
   END_VAR
BEGIN

REGION Network 1 (SCL)
   IF NOT "AHUAlarms".Summary.FrostAlarm[#iUnitID] AND NOT "AHUAlarms".Summary.BlockingAlarm[#iUnitID] THEN
       // Statement section IF
       #cTargetState := 7;
       #cHeatingRegState := #cHeatingRegCfg;
       #cCoolingRegState := #cCoolingRegCfg;
       #cIAQRegState := #cHeatingRegCfg;
       #cHeatingRegState := #cHeatingRegCfg;


   END_IF;
END_REGION
END_FUNCTION

FUNCTION "AHURegsAndTargetStatesInEconomyOpMode" : Void   // FC60031, LAD
{ S7_Optimized_Access := 'TRUE' }
VERSION : 0.1
// Operation Modes                                                 Unit State
// 0                                                                              0=Stopped
// 1=Economy                                                           1=Checking-up  
//                                                                                 2=Preheating
//                                                                                 3=Starting 
//                                                                                 4=RecirculatingOperation (Protection)
//                                                                                 5=Sustained Mode (Economy)
//                                                                                 Not 6=Sustained Mode (PreComfort setpoints) 
//                                                                                 Not 7=Comfort  operation
//                                                                                 Not 8=Night Cooling
//                                                                                 9=Stopping
//                                                                                 10=Blocking
//                                                                                 11=FrostProtecting
// stored: AutoNumber false, IsIECCheckEnabled false, SetENOAutomatically false, UDAEnableTagReadback false
   VAR_INPUT
      iUnitID : Int;
      cActualOpMode : Byte;
      cHeatingRegCfg : Byte;
      cCoolingRegCfg : Byte;
      cIAQRegCfg : Byte;
      cBuildingdPRegCfg : Byte;
   END_VAR
   VAR_OUTPUT
      cTargetState : Byte;
      cHeatingRegState : Byte;
      cCoolingRegState : Byte;
      cIAQRegState : Byte;
      cBuildingdPRegState : Byte;
   END_VAR
   VAR_TEMP
      SHTargetState : Int;
      SCTargetState : Int;
      SIAQTargetState : Int;
      SdPTargetState : Int;
   END_VAR
BEGIN

REGION Network 1: Sustained Heating
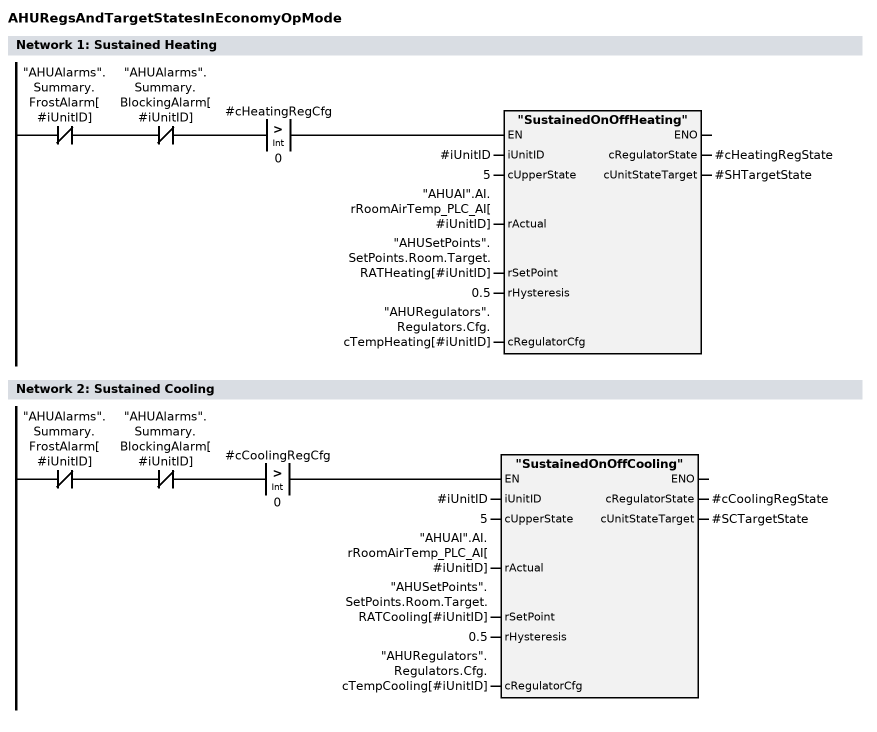
   RUNG wire#powerrail
      I_Contact( "AHUAlarms".Summary.FrostAlarm[#iUnitID] )
      I_Contact( "AHUAlarms".Summary.BlockingAlarm[#iUnitID] )
      { S7_Templates := "SrcType := Int" } GT_Contact(in1 := #cHeatingRegCfg, in2 := 0)
      "SustainedOnOffHeating"(iUnitID := #iUnitID, cUpperState := 5, rActual := "AHUAI".AI.rRoomAirTemp_PLC_AI[#iUnitID], rSetPoint := "AHUSetPoints".SetPoints.Room.Target.RATHeating[#iUnitID], rHysteresis := 0.5, cRegulatorCfg := "AHURegulators".Regulators.Cfg.cTempHeating[#iUnitID], cRegulatorState => #cHeatingRegState, cUnitStateTarget => #SHTargetState)
   END_RUNG
   // the same network as SCL:
   IF NOT "AHUAlarms".Summary.FrostAlarm[#iUnitID] AND NOT "AHUAlarms".Summary.BlockingAlarm[#iUnitID] AND (#cHeatingRegCfg > 0) THEN
       "SustainedOnOffHeating"(iUnitID := #iUnitID,
                               cUpperState := 5,
                               rActual := "AHUAI".AI.rRoomAirTemp_PLC_AI[#iUnitID],
                               rSetPoint := "AHUSetPoints".SetPoints.Room.Target.RATHeating[#iUnitID],
                               rHysteresis := 0.5,
                               cRegulatorCfg := "AHURegulators".Regulators.Cfg.cTempHeating[#iUnitID],
                               cRegulatorState => #cHeatingRegState,
                               cUnitStateTarget => #SHTargetState);
   END_IF;
END_REGION

REGION Network 2: Sustained Cooling
   RUNG wire#powerrail
      I_Contact( "AHUAlarms".Summary.FrostAlarm[#iUnitID] )
      I_Contact( "AHUAlarms".Summary.BlockingAlarm[#iUnitID] )
      { S7_Templates := "SrcType := Int" } GT_Contact(in1 := #cCoolingRegCfg, in2 := 0)
      "SustainedOnOffCooling"(iUnitID := #iUnitID, cUpperState := 5, rActual := "AHUAI".AI.rRoomAirTemp_PLC_AI[#iUnitID], rSetPoint := "AHUSetPoints".SetPoints.Room.Target.RATCooling[#iUnitID], rHysteresis := 0.5, cRegulatorCfg := "AHURegulators".Regulators.Cfg.cTempCooling[#iUnitID], cRegulatorState => #cCoolingRegState, cUnitStateTarget => #SCTargetState)
   END_RUNG
   // the same network as SCL:
   IF NOT "AHUAlarms".Summary.FrostAlarm[#iUnitID] AND NOT "AHUAlarms".Summary.BlockingAlarm[#iUnitID] AND (#cCoolingRegCfg > 0) THEN
       "SustainedOnOffCooling"(iUnitID := #iUnitID,
                               cUpperState := 5,
                               rActual := "AHUAI".AI.rRoomAirTemp_PLC_AI[#iUnitID],
                               rSetPoint := "AHUSetPoints".SetPoints.Room.Target.RATCooling[#iUnitID],
                               rHysteresis := 0.5,
                               cRegulatorCfg := "AHURegulators".Regulators.Cfg.cTempCooling[#iUnitID],
                               cRegulatorState => #cCoolingRegState,
                               cUnitStateTarget => #SCTargetState);
   END_IF;
END_REGION

REGION Network 3 (SCL)
   #cTargetState := INT_TO_BYTE(MAX(IN1 := #SHTargetState, IN2 := #SCTargetState));
END_REGION
END_FUNCTION

FUNCTION "SustainedOnOffHeating" : Void   // FC4, FBD
{ S7_Optimized_Access := 'TRUE' }
VERSION : 0.1
// stored: AutoNumber true, IsIECCheckEnabled false, SetENOAutomatically false, UDAEnableTagReadback false
   VAR_INPUT
      iUnitID : Int;
      cUpperState : Byte;
      rActual : Real;
      rSetPoint : Real;
      rHysteresis : Real;
      cRegulatorCfg : Byte;
   END_VAR
   VAR_OUTPUT
      cRegulatorState : Byte;
      cUnitStateTarget : Byte;
   END_VAR
BEGIN

REGION Network 1 (SCL)
   IF #rActual < #rSetPoint - #rHysteresis THEN
       #cUnitStateTarget := #cUpperState;
       #cRegulatorState := #cRegulatorCfg;
   ELSIF #cUnitStateTarget = #cUpperState AND #rActual > #rSetPoint + #rHysteresis THEN
       #cUnitStateTarget := 0;
       #cRegulatorState := 0;
   ELSE
       #cUnitStateTarget := 0;
       #cRegulatorState := 0;
   END_IF;
END_REGION
END_FUNCTION

FUNCTION "SustainedOnOffCooling" : Void   // FC7, FBD
{ S7_Optimized_Access := 'TRUE' }
VERSION : 0.1
// stored: AutoNumber true, IsIECCheckEnabled false, SetENOAutomatically false, UDAEnableTagReadback false
   VAR_INPUT
      iUnitID : Int;
      cUpperState : Byte;
      rActual : Real;
      rSetPoint : Real;
      rHysteresis : Real;
      cRegulatorCfg : Byte;
   END_VAR
   VAR_OUTPUT
      cRegulatorState : Byte;
      cUnitStateTarget : Byte;
   END_VAR
BEGIN

REGION Network 1 (SCL)
   IF #rActual > #rSetPoint + #rHysteresis THEN
       #cUnitStateTarget := #cUpperState;
       #cRegulatorState := #cRegulatorCfg;
   ELSIF #cUnitStateTarget = #cUpperState AND #rActual < #rSetPoint - #rHysteresis THEN
       #cUnitStateTarget := 0;
       #cRegulatorState := 0;
   ELSE
       #cUnitStateTarget := 0;
       #cRegulatorState := 0;
   END_IF;
END_REGION
END_FUNCTION

FUNCTION "AHURegsAndTargetStatesInPreComfortOpMode" : Void   // FC60032, LAD
{ S7_Optimized_Access := 'TRUE' }
VERSION : 0.1
// Operation Modes                                                 Unit State
// 0                                                                             0=Stopped
// 1                                                                             1=Checking-up  
// 2 PreComfort                                                        2=Preheating
//                                                                                 3=Starting 
//                                                                                 4=RecirculatingOperation (Protection)
//                                                                                 5=Sustained Mode (Economy)
//                                                                                 6=Sustained Mode (PreComfort setpoints) 
//                                                                                 Not 7=Comfort  operation
//                                                                                 Not 8=Night Cooling
//                                                                                 9=Stopping
//                                                                                 10=Blocking
//                                                                                 11=FrostProtecting
// stored: AutoNumber false, IsIECCheckEnabled false, SetENOAutomatically false, UDAEnableTagReadback false
   VAR_INPUT
      iUnitID : Int;
      cActualOpMode : Byte;
      cHeatingRegCfg : Byte;
      cCoolingRegCfg : Byte;
      cIAQRegCfg : Byte;
      cBuildingdPRegCfg : Byte;
   END_VAR
   VAR_OUTPUT
      cTargetState : Byte;
      cHeatingRegState : Byte;
      cCoolingRegState : Byte;
      cIAQRegState : Byte;
      cBuildingdPRegState : Byte;
   END_VAR
   VAR_TEMP
      SHTargetState : Byte;
      SCTargetState : Byte;
      SIAQTargetState : Byte;
      SdPTargetState : Byte;
   END_VAR
BEGIN

REGION Network 1: Sustained Heating
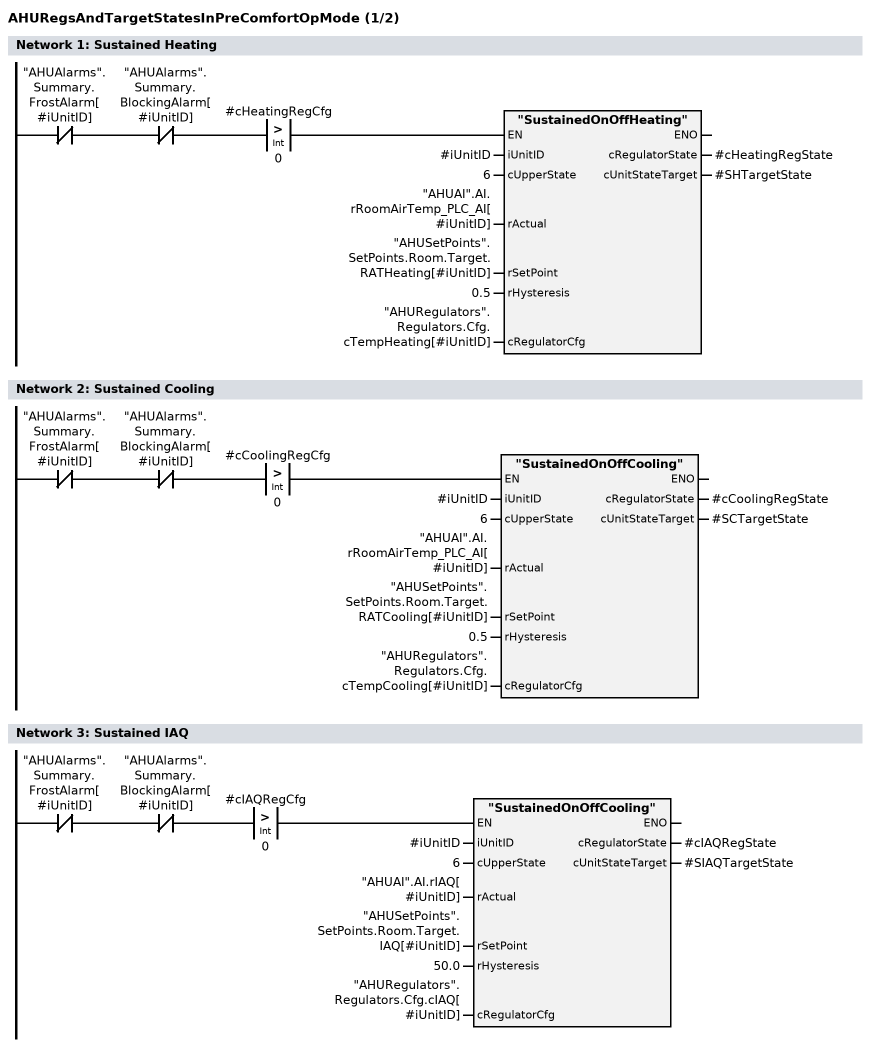
   RUNG wire#powerrail
      I_Contact( "AHUAlarms".Summary.FrostAlarm[#iUnitID] )
      I_Contact( "AHUAlarms".Summary.BlockingAlarm[#iUnitID] )
      { S7_Templates := "SrcType := Int" } GT_Contact(in1 := #cHeatingRegCfg, in2 := 0)
      "SustainedOnOffHeating"(iUnitID := #iUnitID, cUpperState := 6, rActual := "AHUAI".AI.rRoomAirTemp_PLC_AI[#iUnitID], rSetPoint := "AHUSetPoints".SetPoints.Room.Target.RATHeating[#iUnitID], rHysteresis := 0.5, cRegulatorCfg := "AHURegulators".Regulators.Cfg.cTempHeating[#iUnitID], cRegulatorState => #cHeatingRegState, cUnitStateTarget => #SHTargetState)
   END_RUNG
   // the same network as SCL:
   IF NOT "AHUAlarms".Summary.FrostAlarm[#iUnitID] AND NOT "AHUAlarms".Summary.BlockingAlarm[#iUnitID] AND (#cHeatingRegCfg > 0) THEN
       "SustainedOnOffHeating"(iUnitID := #iUnitID,
                               cUpperState := 6,
                               rActual := "AHUAI".AI.rRoomAirTemp_PLC_AI[#iUnitID],
                               rSetPoint := "AHUSetPoints".SetPoints.Room.Target.RATHeating[#iUnitID],
                               rHysteresis := 0.5,
                               cRegulatorCfg := "AHURegulators".Regulators.Cfg.cTempHeating[#iUnitID],
                               cRegulatorState => #cHeatingRegState,
                               cUnitStateTarget => #SHTargetState);
   END_IF;
END_REGION

REGION Network 2: Sustained Cooling
   RUNG wire#powerrail
      I_Contact( "AHUAlarms".Summary.FrostAlarm[#iUnitID] )
      I_Contact( "AHUAlarms".Summary.BlockingAlarm[#iUnitID] )
      { S7_Templates := "SrcType := Int" } GT_Contact(in1 := #cCoolingRegCfg, in2 := 0)
      "SustainedOnOffCooling"(iUnitID := #iUnitID, cUpperState := 6, rActual := "AHUAI".AI.rRoomAirTemp_PLC_AI[#iUnitID], rSetPoint := "AHUSetPoints".SetPoints.Room.Target.RATCooling[#iUnitID], rHysteresis := 0.5, cRegulatorCfg := "AHURegulators".Regulators.Cfg.cTempCooling[#iUnitID], cRegulatorState => #cCoolingRegState, cUnitStateTarget => #SCTargetState)
   END_RUNG
   // the same network as SCL:
   IF NOT "AHUAlarms".Summary.FrostAlarm[#iUnitID] AND NOT "AHUAlarms".Summary.BlockingAlarm[#iUnitID] AND (#cCoolingRegCfg > 0) THEN
       "SustainedOnOffCooling"(iUnitID := #iUnitID,
                               cUpperState := 6,
                               rActual := "AHUAI".AI.rRoomAirTemp_PLC_AI[#iUnitID],
                               rSetPoint := "AHUSetPoints".SetPoints.Room.Target.RATCooling[#iUnitID],
                               rHysteresis := 0.5,
                               cRegulatorCfg := "AHURegulators".Regulators.Cfg.cTempCooling[#iUnitID],
                               cRegulatorState => #cCoolingRegState,
                               cUnitStateTarget => #SCTargetState);
   END_IF;
END_REGION

REGION Network 3: Sustained IAQ
   RUNG wire#powerrail
      I_Contact( "AHUAlarms".Summary.FrostAlarm[#iUnitID] )
      I_Contact( "AHUAlarms".Summary.BlockingAlarm[#iUnitID] )
      { S7_Templates := "SrcType := Int" } GT_Contact(in1 := #cIAQRegCfg, in2 := 0)
      "SustainedOnOffCooling"(iUnitID := #iUnitID, cUpperState := 6, rActual := "AHUAI".AI.rIAQ[#iUnitID], rSetPoint := "AHUSetPoints".SetPoints.Room.Target.IAQ[#iUnitID], rHysteresis := 50.0, cRegulatorCfg := "AHURegulators".Regulators.Cfg.cIAQ[#iUnitID], cRegulatorState => #cIAQRegState, cUnitStateTarget => #SIAQTargetState)
   END_RUNG
   // the same network as SCL:
   IF NOT "AHUAlarms".Summary.FrostAlarm[#iUnitID] AND NOT "AHUAlarms".Summary.BlockingAlarm[#iUnitID] AND (#cIAQRegCfg > 0) THEN
       "SustainedOnOffCooling"(iUnitID := #iUnitID,
                               cUpperState := 6,
                               rActual := "AHUAI".AI.rIAQ[#iUnitID],
                               rSetPoint := "AHUSetPoints".SetPoints.Room.Target.IAQ[#iUnitID],
                               rHysteresis := 50.0,
                               cRegulatorCfg := "AHURegulators".Regulators.Cfg.cIAQ[#iUnitID],
                               cRegulatorState => #cIAQRegState,
                               cUnitStateTarget => #SIAQTargetState);
   END_IF;
END_REGION

REGION Network 4: Sustained BuildingdP
   // !!!!Додати опрацьовку Сили вітриу з погодної станції
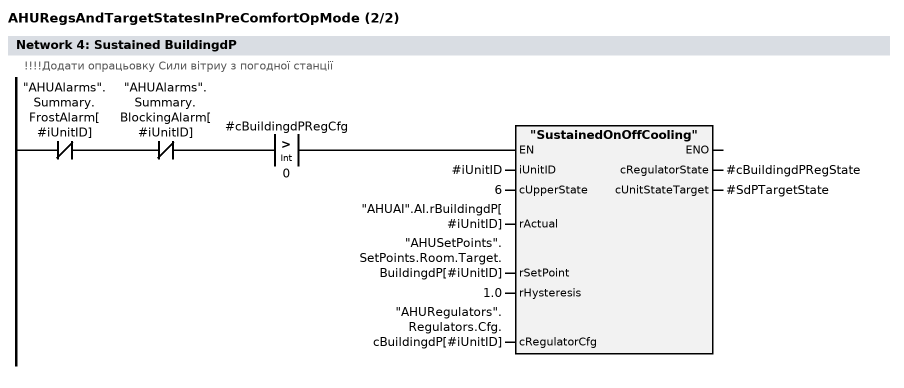
   RUNG wire#powerrail
      I_Contact( "AHUAlarms".Summary.FrostAlarm[#iUnitID] )
      I_Contact( "AHUAlarms".Summary.BlockingAlarm[#iUnitID] )
      { S7_Templates := "SrcType := Int" } GT_Contact(in1 := #cBuildingdPRegCfg, in2 := 0)
      "SustainedOnOffCooling"(iUnitID := #iUnitID, cUpperState := 6, rActual := "AHUAI".AI.rBuildingdP[#iUnitID], rSetPoint := "AHUSetPoints".SetPoints.Room.Target.BuildingdP[#iUnitID], rHysteresis := 1.0, cRegulatorCfg := "AHURegulators".Regulators.Cfg.cBuildingdP[#iUnitID], cRegulatorState => #cBuildingdPRegState, cUnitStateTarget => #SdPTargetState)
   END_RUNG
   // the same network as SCL:
   IF NOT "AHUAlarms".Summary.FrostAlarm[#iUnitID] AND NOT "AHUAlarms".Summary.BlockingAlarm[#iUnitID] AND (#cBuildingdPRegCfg > 0) THEN
       "SustainedOnOffCooling"(iUnitID := #iUnitID,
                               cUpperState := 6,
                               rActual := "AHUAI".AI.rBuildingdP[#iUnitID],
                               rSetPoint := "AHUSetPoints".SetPoints.Room.Target.BuildingdP[#iUnitID],
                               rHysteresis := 1.0,
                               cRegulatorCfg := "AHURegulators".Regulators.Cfg.cBuildingdP[#iUnitID],
                               cRegulatorState => #cBuildingdPRegState,
                               cUnitStateTarget => #SdPTargetState);
   END_IF;
END_REGION

REGION Network 5 (SCL)
   #SHTargetState := MAX(IN1 := #SHTargetState, IN2 := #SCTargetState);
   #SIAQTargetState := MAX(IN1 := #SIAQTargetState, IN2 := #SdPTargetState);
   #cTargetState := MAX(IN1 := #SIAQTargetState, IN2 := #SHTargetState);
END_REGION
END_FUNCTION

FUNCTION "AHURegsAndTargetStatesInProtectionOpMode" : Void   // FC60034, LAD
{ S7_Optimized_Access := 'TRUE' }
VERSION : 0.1
// Operation Modes                                                 Unit State
// 0=Protection                                                         0=Stopped
//                                                                                 1=Checking-up  
//                                                                                 2=Preheating
//                                                                                 3=Starting 
//                                                                                 4=RecirculatingOperation (Protection)
//                                                                                 Not 5=Sustained Mode (Economy)
//                                                                                 Not 6=Sustained Mode (PreComfort setpoints) 
//                                                                                 Not 7=Comfort  operation
//                                                                                 Not 8=Night Cooling
//                                                                                 9=Stopping
//                                                                                 10=Blocking
//                                                                                 11=FrostProtecting
// stored: AutoNumber false, IsIECCheckEnabled false, SetENOAutomatically false, UDAEnableTagReadback false
   VAR_INPUT
      iUnitID : Int;
      cActualOpMode : Byte;
      cHeatingRegCfg : Byte;
      cCoolingRegCfg : Byte;
      cIAQRegCfg : Byte;
      cBuildingdPRegCfg : Byte;
   END_VAR
   VAR_OUTPUT
      cTargetState : Byte;
      cHeatingRegState : Byte;
      cCoolingRegState : Byte;
      cIAQRegState : Byte;
      cBuildingdPRegState : Byte;
   END_VAR
   VAR_TEMP
      cSHTargetState : Byte;
      cSCTargetState : Byte;
      cSIAQTargetState : Byte;
      cSdPTargetState : Byte;
   END_VAR
BEGIN

REGION Network 1
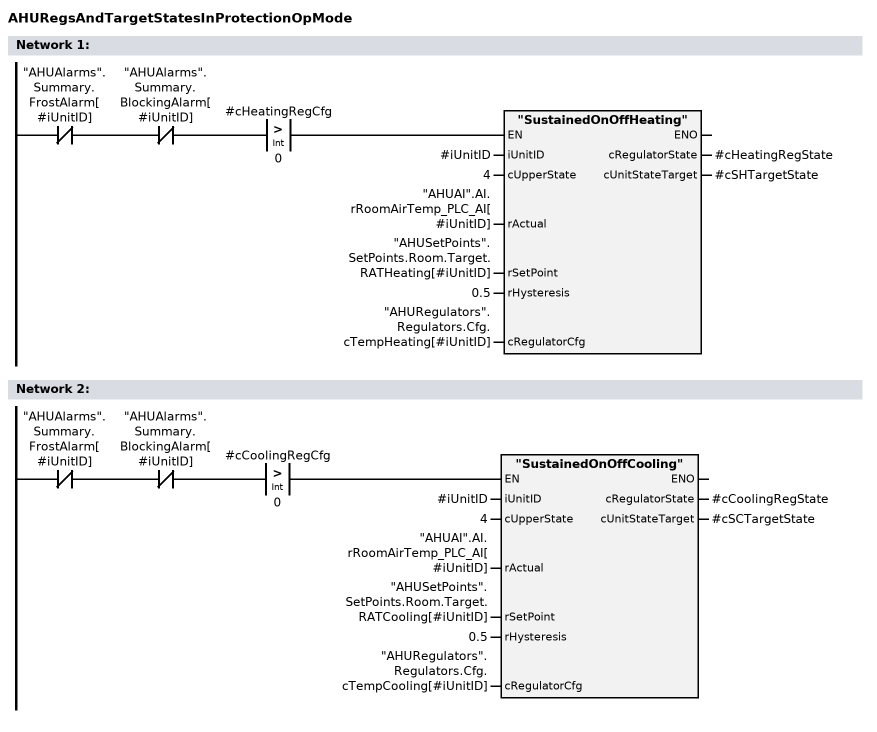
   RUNG wire#powerrail
      I_Contact( "AHUAlarms".Summary.FrostAlarm[#iUnitID] )
      I_Contact( "AHUAlarms".Summary.BlockingAlarm[#iUnitID] )
      { S7_Templates := "SrcType := Int" } GT_Contact(in1 := #cHeatingRegCfg, in2 := 0)
      "SustainedOnOffHeating"(iUnitID := #iUnitID, cUpperState := 4, rActual := "AHUAI".AI.rRoomAirTemp_PLC_AI[#iUnitID], rSetPoint := "AHUSetPoints".SetPoints.Room.Target.RATHeating[#iUnitID], rHysteresis := 0.5, cRegulatorCfg := "AHURegulators".Regulators.Cfg.cTempHeating[#iUnitID], cRegulatorState => #cHeatingRegState, cUnitStateTarget => #cSHTargetState)
   END_RUNG
   // the same network as SCL:
   IF NOT "AHUAlarms".Summary.FrostAlarm[#iUnitID] AND NOT "AHUAlarms".Summary.BlockingAlarm[#iUnitID] AND (#cHeatingRegCfg > 0) THEN
       "SustainedOnOffHeating"(iUnitID := #iUnitID,
                               cUpperState := 4,
                               rActual := "AHUAI".AI.rRoomAirTemp_PLC_AI[#iUnitID],
                               rSetPoint := "AHUSetPoints".SetPoints.Room.Target.RATHeating[#iUnitID],
                               rHysteresis := 0.5,
                               cRegulatorCfg := "AHURegulators".Regulators.Cfg.cTempHeating[#iUnitID],
                               cRegulatorState => #cHeatingRegState,
                               cUnitStateTarget => #cSHTargetState);
   END_IF;
END_REGION

REGION Network 2
   RUNG wire#powerrail
      I_Contact( "AHUAlarms".Summary.FrostAlarm[#iUnitID] )
      I_Contact( "AHUAlarms".Summary.BlockingAlarm[#iUnitID] )
      { S7_Templates := "SrcType := Int" } GT_Contact(in1 := #cCoolingRegCfg, in2 := 0)
      "SustainedOnOffCooling"(iUnitID := #iUnitID, cUpperState := 4, rActual := "AHUAI".AI.rRoomAirTemp_PLC_AI[#iUnitID], rSetPoint := "AHUSetPoints".SetPoints.Room.Target.RATCooling[#iUnitID], rHysteresis := 0.5, cRegulatorCfg := "AHURegulators".Regulators.Cfg.cTempCooling[#iUnitID], cRegulatorState => #cCoolingRegState, cUnitStateTarget => #cSCTargetState)
   END_RUNG
   // the same network as SCL:
   IF NOT "AHUAlarms".Summary.FrostAlarm[#iUnitID] AND NOT "AHUAlarms".Summary.BlockingAlarm[#iUnitID] AND (#cCoolingRegCfg > 0) THEN
       "SustainedOnOffCooling"(iUnitID := #iUnitID,
                               cUpperState := 4,
                               rActual := "AHUAI".AI.rRoomAirTemp_PLC_AI[#iUnitID],
                               rSetPoint := "AHUSetPoints".SetPoints.Room.Target.RATCooling[#iUnitID],
                               rHysteresis := 0.5,
                               cRegulatorCfg := "AHURegulators".Regulators.Cfg.cTempCooling[#iUnitID],
                               cRegulatorState => #cCoolingRegState,
                               cUnitStateTarget => #cSCTargetState);
   END_IF;
END_REGION

REGION Network 3 (SCL)
   #cTargetState := MAX(IN1 := #cSHTargetState, IN2 := #cSCTargetState);
END_REGION
END_FUNCTION

FUNCTION "AHURegsCtrl_1" : Void   // FC60035, LAD
{ S7_Optimized_Access := 'TRUE' }
VERSION : 0.1
// Operation Modes                                                 Unit State
// 0=Protection                                                         0=Stopped
// 1=Economy                                                           1=Checking-up  
// 2=PreComfort                                                       2=Preheating
// 3=Comfor                                                              3=Starting 
// 4=Auto(Scheduler)                                              4=RecirculatingOperation (Protection)
//                                                                                 5=Sustained Mode (Economy setpoints)
//                                                                                 6=Sustained Mode (PreComfort setpoints) 
//                                                                                 7=Comfort  operation
//                                                                                 8=Stopping
//                                                                                 9=Blocking
// stored: AutoNumber false, IsIECCheckEnabled false, SetENOAutomatically false, UDAEnableTagReadback false
   VAR_INPUT
      iUnitID : Int;
      cActualOpMode : Byte;
      cHeatingRegCfg : Byte;
      cCoolingRegCfg : Byte;
      cIAQRegCfg : Byte;
      cBuildingdPRegCfg : Byte;
      xOtherBlockingAlarm : Bool;
      xFrostProtBlocking : Bool;
   END_VAR
   VAR_OUTPUT
      cTargetState : Byte;
      cHeatingRegState : Byte;
      cCoolingRegState : Byte;
      cIAQRegState : Byte;
      cBuildingdPRegState : Byte;
   END_VAR
   VAR_TEMP
      cActualOpModeSequence : Byte;   // Поточний цикл
   END_VAR
BEGIN

REGION Network 1 (SCL)
   IF #xFrostProtBlocking THEN
       // Frost protection
       #cTargetState := 11;
   ELSIF #xOtherBlockingAlarm THEN
       // Blocking Alarm
       #cTargetState := 10;
   ELSE
       CASE #cActualOpMode OF
           0:  // Protection 
               "AHURegsAndTargetStatesInProtectionOpMode"(iUnitID:=#iUnitID,
                                                          cActualOpMode:=#cActualOpMode,
                                                          cHeatingRegCfg:=#cHeatingRegCfg,
                                                          cCoolingRegCfg:=#cCoolingRegCfg,
                                                          cIAQRegCfg:=#cIAQRegCfg,
                                                          cBuildingdPRegCfg:=#cBuildingdPRegCfg,
                                                          cTargetState=>#cTargetState,
                                                          cHeatingRegState=>#cHeatingRegState,
                                                          cCoolingRegState=>#cCoolingRegState,
                                                          cIAQRegState=>#cIAQRegState,
                                                          cBuildingdPRegState=>#cBuildingdPRegState);

           1:  // Economy
               "AHURegsAndTargetStatesInEconomyOpMode"(iUnitID:=#iUnitID,
                                                       cActualOpMode:=#cActualOpMode,
                                                       cHeatingRegCfg:=#cHeatingRegCfg,
                                                       cCoolingRegCfg:=#cCoolingRegCfg,
                                                       cIAQRegCfg:=#cIAQRegCfg,
                                                       cBuildingdPRegCfg:=#cBuildingdPRegCfg,
                                                       cTargetState=>#cTargetState,
                                                       cHeatingRegState=>#cHeatingRegState,
                                                       cCoolingRegState=>#cCoolingRegState,
                                                       cIAQRegState=>#cIAQRegState,
                                                       cBuildingdPRegState=>#cBuildingdPRegState);
           2: // PreComfort
               "AHURegsAndTargetStatesInPreComfortOpMode"(iUnitID:=#iUnitID,
                                                          cActualOpMode:=#cActualOpMode,
                                                          cHeatingRegCfg:=#cHeatingRegCfg,
                                                          cCoolingRegCfg:=#cCoolingRegCfg,
                                                          cIAQRegCfg:=#cIAQRegCfg,
                                                          cBuildingdPRegCfg:=#cBuildingdPRegCfg,
                                                          cTargetState=>#cTargetState,
                                                          cHeatingRegState=>#cHeatingRegState,
                                                          cCoolingRegState=>#cCoolingRegState,
                                                          cIAQRegState=>#cIAQRegState,
                                                          cBuildingdPRegState=>#cBuildingdPRegState);
           ELSE  //Comfort
               "AHURegsAndTargetStatesInComfortOpMode"(iUnitID:=#iUnitID,
                                                       cActualOpMode:=#cActualOpMode,
                                                       cHeatingRegCfg:=#cHeatingRegCfg,
                                                       cCoolingRegCfg:=#cCoolingRegCfg,
                                                       cIAQRegCfg:=#cIAQRegCfg,
                                                       cBuildingdPRegCfg:=#cBuildingdPRegCfg,
                                                       cTargetState=>#cTargetState,
                                                       cHeatingRegState=>#cHeatingRegState,
                                                       cCoolingRegState=>#cCoolingRegState,
                                                       cIAQRegState=>#cIAQRegState,
                                                       cBuildingdPRegState=>#cBuildingdPRegState);
       END_CASE;
       ;
   END_IF;
END_REGION
END_FUNCTION

FUNCTION "AHUSPCtrl" : Void   // FC60003, LAD
{ S7_Optimized_Access := 'TRUE' }
VERSION : 0.1
// stored: AutoNumber false, IsIECCheckEnabled false, SetENOAutomatically false, UDAEnableTagReadback false
   VAR_INPUT
      iUnitID : Int;
      rProtTempHeating : Real;
      rEconTempHeating : Real;
      rPreComfTempHeating : Real;
      rComfTempHeating : Real;
      rComfTempCooling : Real;
      rPreComfTempCooling : Real;
      rEconTempCooling : Real;
      rProtTempCooling : Real;
      rProtIAQ : Real;
      rEconIAQ : Real;
      rPreComfIAQ : Real;
      rComfIAQ : Real;
      rProtdP : Real;
      rEcondP : Real;
      rPreComfdP : Real;
      rComfdP : Real;
   END_VAR
   VAR_OUTPUT
      rActualTempHeating : Real;
      rActualTempCooling : Real;
      rActualIAQ : Real;
      rActualdP : Real;
   END_VAR
   VAR_TEMP
      iTargetUnitMode_old : Int;
      xResetActualOperationMode : Bool;
      iActualUnitMode_old : Int;
      xResetTargetSetpoints : Bool;
   END_VAR
BEGIN

REGION Network 1 (SCL)
   // Redefine Target Setpoints
   IF "AHUOpModes".OpModes.cActual[#iUnitID] = "AHUOpModes".OpModes.cTarget[#iUnitID] THEN // !!!Змінити на PrevOpMode
       // Statement section IF
       CASE "AHUOpModes".OpModes.cActual[#iUnitID] OF
           0:  // Protection
               "AHUSetPoints".SetPoints.Room.Target.RATHeating[#iUnitID] := #rProtTempHeating;
               "AHUSetPoints".SetPoints.Room.Target.RATCooling[#iUnitID] := #rProtTempCooling;
               "AHUSetPoints".SetPoints.Room.Target.IAQ[#iUnitID] := #rProtIAQ;
               "AHUSetPoints".SetPoints.Room.Target.BuildingdP[#iUnitID] := #rProtdP;
           1:  // Economy
               "AHUSetPoints".SetPoints.Room.Target.RATHeating[#iUnitID] := #rEconTempHeating;
               "AHUSetPoints".SetPoints.Room.Target.RATCooling[#iUnitID] := #rEconTempCooling;
               "AHUSetPoints".SetPoints.Room.Target.IAQ[#iUnitID] := #rEconIAQ;
               "AHUSetPoints".SetPoints.Room.Target.BuildingdP[#iUnitID] := #rEcondP;
           2: // Precomfort
               "AHUSetPoints".SetPoints.Room.Target.RATHeating[#iUnitID] := #rPreComfTempHeating;
               "AHUSetPoints".SetPoints.Room.Target.RATCooling[#iUnitID] := #rPreComfTempCooling;
               "AHUSetPoints".SetPoints.Room.Target.IAQ[#iUnitID] := #rPreComfIAQ;
               "AHUSetPoints".SetPoints.Room.Target.BuildingdP[#iUnitID] := #rPreComfdP;
           ELSE  // Statement section ELSE
               "AHUSetPoints".SetPoints.Room.Target.RATHeating[#iUnitID] := #rComfTempHeating;
               "AHUSetPoints".SetPoints.Room.Target.RATCooling[#iUnitID] := #rComfTempCooling;
               "AHUSetPoints".SetPoints.Room.Target.IAQ[#iUnitID] := #rComfIAQ;
               "AHUSetPoints".SetPoints.Room.Target.BuildingdP[#iUnitID] := #rComfdP;
       END_CASE;
       ;
   END_IF;
END_REGION

REGION Network 2 (SCL): Smoothing Actual Setpoints
   IF 1 THEN
       #rActualTempHeating := "AHUSetPoints".SetPoints.Room.Target.RATHeating[#iUnitID];
       #rActualTempCooling := "AHUSetPoints".SetPoints.Room.Target.RATCooling[#iUnitID];
       #rActualIAQ := "AHUSetPoints".SetPoints.Room.Target.IAQ[#iUnitID];
       #rActualdP := "AHUSetPoints".SetPoints.Room.Target.BuildingdP[#iUnitID];
   END_IF;
END_REGION
END_FUNCTION

FUNCTION "HVACSeason" : Void   // FC60020, LAD
{ S7_Optimized_Access := 'TRUE' }
VERSION : 0.1
// stored: AutoNumber false, IsIECCheckEnabled false, SetENOAutomatically false, UDAEnableTagReadback false
BEGIN
END_FUNCTION

DATA_BLOCK "DL_Counter_1"   // DB51052
{ S7_Optimized_Access := 'TRUE' }
// stored: AutoNumber false, DBAccessibleFromOPCUA true, InstanceOfName IEC_COUNTER, OfSystemLibElement IEC_COUNTER, OfSystemLibVersion 1.0
"IEC_COUNTER"
   // VAR RETAIN
   //    CU : Bool;
   //    CD : Bool;
   //    R : Bool;
   //    LD : Bool;
   //    QU : Bool;
   //    QD : Bool;
   //    PV : Int;
   //    CV : Int;
   // END_VAR
BEGIN
END_DATA_BLOCK

DATA_BLOCK "DL_Counter_2"   // DB51053
{ S7_Optimized_Access := 'TRUE' }
// stored: AutoNumber false, DBAccessibleFromOPCUA true, InstanceOfName IEC_COUNTER, OfSystemLibElement IEC_COUNTER, OfSystemLibVersion 1.0
"IEC_COUNTER"
   // VAR RETAIN
   //    CU : Bool;
   //    CD : Bool;
   //    R : Bool;
   //    LD : Bool;
   //    QU : Bool;
   //    QD : Bool;
   //    PV : Int;
   //    CV : Int;
   // END_VAR
BEGIN
END_DATA_BLOCK

DATA_BLOCK "DL_Timer_1_DB"   // DB51054
{ S7_Optimized_Access := 'TRUE' }
// stored: AutoNumber false, DBAccessibleFromOPCUA true, InstanceOfName IEC_TIMER, OfSystemLibElement IEC_TIMER, OfSystemLibVersion 1.0
"IEC_TIMER"
   // VAR
   //    PT : Time;
   //    ET { ExternalWritable := 'False'} : Time;
   //    IN : Bool;
   //    Q { ExternalWritable := 'False'} : Bool;
   // END_VAR
BEGIN
END_DATA_BLOCK

DATA_BLOCK "DL_Timer_2_DB"   // DB51055
{ S7_Optimized_Access := 'TRUE' }
// stored: AutoNumber false, DBAccessibleFromOPCUA true, InstanceOfName IEC_TIMER, OfSystemLibElement IEC_TIMER, OfSystemLibVersion 1.0
"IEC_TIMER"
   // VAR
   //    PT : Time;
   //    ET { ExternalWritable := 'False'} : Time;
   //    IN : Bool;
   //    Q { ExternalWritable := 'False'} : Bool;
   // END_VAR
BEGIN
END_DATA_BLOCK

